LIN {X 0,Y 197.336,Z 414.265,A -85,B 0,C 180,E1 -21920.386,E2 -21920.386} C_VEL
LIN {X 0,Y 196.513,Z 412.639,A -85,B 0,C 180,E1 -21920.854,E2 -21920.854} C_VEL
LIN {X 0,Y 194.043,Z 410.71,A -85,B 0,C 180,E1 -21922.116,E2 -21922.116} C_VEL
LIN {X 0,Y 192.76,Z 408.182,A -85,B 0,C 180,E1 -21922.91,E2 -21922.91} C_VEL
LIN {X 0,Y 192.565,Z 407.12,A -85,B 0,C 180,E1 -21923.107,E2 -21923.107} C_VEL
LIN {X 0,Y 192.604,Z 407.109,A -85,B 0,C 180,E1 -21927.061,E2 -21927.061} C_VEL
LIN {X 0,Y 192.618,Z 407.106,A -85,B 0,C 180,E1 -21931.684,E2 -21931.684} C_VEL
LIN {X 0,Y 192.669,Z 407.096,A -85,B 0,C 180,E1 -21936.343,E2 -21936.343} C_VEL
LIN {X 0,Y 192.693,Z 407.092,A -85,B 0,C 180,E1 -21941.491,E2 -21941.491} C_VEL
LIN {X 0,Y 192.732,Z 407.089,A -85,B 0,C 180,E1 -21945.211,E2 -21945.211} C_VEL
LIN {X 0,Y 192.944,Z 407.006,A -85,B 0,C 180,E1 -21949.566,E2 -21949.566} C_VEL
LIN {X 0,Y 192.953,Z 407.069,A -85,B 0,C 180,E1 -21953.726,E2 -21953.726} C_VEL
LIN {X 0,Y 193.204,Z 407.021,A -85,B 0,C 180,E1 -21957.915,E2 -21957.915} C_VEL
LIN {X 0,Y 193.404,Z 407.012,A -85,B 0,C 180,E1 -21959.999,E2 -21959.999} C_VEL
LIN {X 0,Y 192.929,Z 407.057,A -85,B 0,C 180,E1 -21964.177,E2 -21964.177} C_VEL
LIN {X 0,Y 193.017,Z 407.052,A -85,B 0,C 180,E1 -21968.374,E2 -21968.374} C_VEL
LIN {X 0,Y 192.77,Z 407.094,A -85,B 0,C 180,E1 -21972.635,E2 -21972.635} C_VEL
LIN {X 0,Y 192.692,Z 407.097,A -85,B 0,C 180,E1 -21978.508,E2 -21978.508} C_VEL
LIN {X 0,Y 192.648,Z 407.204,A -85,B 0,C 180,E1 -21982.947,E2 -21982.947} C_VEL
LIN {X 0,Y 195.501,Z 414.864,A -85,B 0,C 180,E1 -21987.715,E2 -21987.715} C_VEL
LIN {X 0,Y 201.405,Z 424.233,A -85,B 0,C 180,E1 -21990.831,E2 -21990.831} C_VEL
LIN {X 0,Y 205.353,Z 430.73,A -85,B 0,C 180,E1 -21992.69,E2 -21992.69} C_VEL
LIN {X 0,Y 209.382,Z 437.854,A -85,B 0,C 180,E1 -21994.468,E2 -21994.468} C_VEL
LIN {X 0,Y 212.955,Z 444.606,A -85,B 0,C 180,E1 -21995.959,E2 -21995.959} C_VEL
LIN {X 0,Y 217.953,Z 454.685,A -85,B 0,C 180,E1 -21997.928,E2 -21997.928} C_VEL
LIN {X 0,Y 223.379,Z 466.674,A -85,B 0,C 180,E1 -21999.942,E2 -21999.942} C_VEL
LIN {X 0,Y 228.391,Z 479.658,A -85,B 0,C 180,E1 -22001.743,E2 -22001.743} C_VEL
LIN {X 0,Y 229.336,Z 493.154,A -85,B 0,C 180,E1 -22002.532,E2 -22002.532} C_VEL
LIN {X 0,Y 229.333,Z 498.97,A -85,B 0,C 180,E1 -22002.774,E2 -22002.774} C_VEL
LIN {X 0,Y 226.311,Z 518.591,A -85,B 0,C 180,E1 -22002.905,E2 -22002.905} C_VEL
LIN {X 0,Y 226.123,Z 524.463,A -85,B 0,C 180,E1 -22003.109,E2 -22003.109} C_VEL
LIN {X 0,Y 222.374,Z 588.724,A -85,B 0,C 180,E1 -22004.997,E2 -22004.997} C_VEL
LIN {X 0,Y 220.722,Z 604.246,A -85,B 0,C 180,E1 -22005.693,E2 -22005.693} C_VEL
LIN {X 0,Y 218.207,Z 619.257,A -85,B 0,C 180,E1 -22006.652,E2 -22006.652} C_VEL
LIN {X 0,Y 215.296,Z 632.891,A -85,B 0,C 180,E1 -22007.838,E2 -22007.838} C_VEL
LIN {X 0,Y 211.683,Z 646.439,A -85,B 0,C 180,E1 -22009.341,E2 -22009.341} C_VEL
LIN {X 0,Y 207.749,Z 658.936,A -85,B 0,C 180,E1 -22011.084,E2 -22011.084} C_VEL
LIN {X 0,Y 204.93,Z 667.258,A -85,B 0,C 180,E1 -22012.503,E2 -22012.503} C_VEL
LIN {X 0,Y 200.796,Z 679.406,A -85,B 0,C 180,E1 -22015.031,E2 -22015.031} C_VEL
LIN {X 0,Y 196.253,Z 691.345,A -85,B 0,C 180,E1 -22018.115,E2 -22018.115} C_VEL
LIN {X 0,Y 192.23,Z 702.077,A -85,B 0,C 180,E1 -22021.622,E2 -22021.622} C_VEL
LIN {X 0,Y 189.098,Z 711.051,A -85,B 0,C 180,E1 -22025.284,E2 -22025.284} C_VEL
LIN {X 0,Y 186.788,Z 718.548,A -85,B 0,C 180,E1 -22029.056,E2 -22029.056} C_VEL
LIN {X 0,Y 185.109,Z 725.529,A -85,B 0,C 180,E1 -22033.456,E2 -22033.456} C_VEL
LIN {X 0,Y 184.507,Z 731.031,A -85,B 0,C 180,E1 -22037.906,E2 -22037.906} C_VEL
LIN {X 0,Y 184.68,Z 734.604,A -85,B 0,C 180,E1 -22041.659,E2 -22041.659} C_VEL
LIN {X 0,Y 185.236,Z 737.321,A -85,B 0,C 180,E1 -22045.647,E2 -22045.647} C_VEL
LIN {X 0,Y 186.173,Z 739.099,A -85,B 0,C 180,E1 -22049.999,E2 -22049.999} C_VEL
LIN {X 0,Y 185.102,Z 739.29,A -85,B 0,C 180,E1 -22054.354,E2 -22054.354} C_VEL
LIN {X 0,Y 184.505,Z 738.486,A -85,B 0,C 180,E1 -22057.961,E2 -22057.961} C_VEL
LIN {X 0,Y 184.298,Z 735.96,A -85,B 0,C 180,E1 -22063.225,E2 -22063.225} C_VEL
LIN {X 0,Y 185.311,Z 732.569,A -85,B 0,C 180,E1 -22067.661,E2 -22067.661} C_VEL
LIN {X 0,Y 187.383,Z 727.977,A -85,B 0,C 180,E1 -22072.027,E2 -22072.027} C_VEL
LIN {X 0,Y 190.614,Z 722.095,A -85,B 0,C 180,E1 -22076.258,E2 -22076.258} C_VEL
LIN {X 0,Y 194.914,Z 714.773,A -85,B 0,C 180,E1 -22080.316,E2 -22080.316} C_VEL
LIN {X 0,Y 200.248,Z 705.81,A -85,B 0,C 180,E1 -22084.161,E2 -22084.161} C_VEL
LIN {X 0,Y 205.88,Z 696.435,A -85,B 0,C 180,E1 -22087.293,E2 -22087.293} C_VEL
LIN {X 0,Y 211.59,Z 686.323,A -85,B 0,C 180,E1 -22089.972,E2 -22089.972} C_VEL
LIN {X 0,Y 217.488,Z 674.798,A -85,B 0,C 180,E1 -22092.418,E2 -22092.418} C_VEL
LIN {X 0,Y 223.387,Z 662.521,A -85,B 0,C 180,E1 -22094.425,E2 -22094.425} C_VEL
LIN {X 0,Y 229.069,Z 649.104,A -85,B 0,C 180,E1 -22096.134,E2 -22096.134} C_VEL
LIN {X 0,Y 233.791,Z 636.023,A -85,B 0,C 180,E1 -22097.431,E2 -22097.431} C_VEL
LIN {X 0,Y 237.121,Z 625.222,A -85,B 0,C 180,E1 -22098.288,E2 -22098.288} C_VEL
LIN {X 0,Y 240.717,Z 610.446,A -85,B 0,C 180,E1 -22099.222,E2 -22099.222} C_VEL
LIN {X 0,Y 243.456,Z 595.214,A -85,B 0,C 180,E1 -22099.904,E2 -22099.904} C_VEL
LIN {X 0,Y 245.117,Z 579.442,A -85,B 0,C 180,E1 -22100.401,E2 -22100.401} C_VEL
LIN {X 0,Y 248.733,Z 529.136,A -85,B 0,C 180,E1 -22101.696,E2 -22101.696} C_VEL
LIN {X 0,Y 247.505,Z 504.831,A -85,B 0,C 180,E1 -22103.33,E2 -22103.33} C_VEL
LIN {X 0,Y 243.68,Z 494.924,A -85,B 0,C 180,E1 -22105.25,E2 -22105.25} C_VEL
LIN {X 0,Y 238.561,Z 483.088,A -85,B 0,C 180,E1 -22108.02,E2 -22108.02} C_VEL
LIN {X 0,Y 234.67,Z 475.032,A -85,B 0,C 180,E1 -22110.329,E2 -22110.329} C_VEL
LIN {X 0,Y 231.739,Z 469.172,A -85,B 0,C 180,E1 -22112.247,E2 -22112.247} C_VEL
LIN {X 0,Y 229.497,Z 464.737,A -85,B 0,C 180,E1 -22113.851,E2 -22113.851} C_VEL
LIN {X 0,Y 225.583,Z 457.444,A -85,B 0,C 180,E1 -22116.991,E2 -22116.991} C_VEL
LIN {X 0,Y 221.261,Z 449.476,A -85,B 0,C 180,E1 -22121.322,E2 -22121.322} C_VEL
LIN {X 0,Y 217.227,Z 441.913,A -85,B 0,C 180,E1 -22127.268,E2 -22127.268} C_VEL
LIN {X 0,Y 215.991,Z 439.112,A -85,B 0,C 180,E1 -22130.327,E2 -22130.327} C_VEL
LIN {X 0,Y 215.609,Z 438.486,A -85,B 0,C 180,E1 -22131.566,E2 -22131.566} C_VEL
LIN {X 0,Y 215.268,Z 438.207,A -85,B 0,C 180,E1 -22140,E2 -22140} C_VEL
LIN {X 0,Y 215.981,Z 438.646,A -85,B 0,C 180,E1 -22142.448,E2 -22142.448} C_VEL
LIN {X 0,Y 217.318,Z 441.615,A -85,B 0,C 180,E1 -22145.801,E2 -22145.801} C_VEL
LIN {X 0,Y 219.851,Z 444.129,A -85,B 0,C 180,E1 -22149.546,E2 -22149.546} C_VEL
LIN {X 0,Y 222.184,Z 447.842,A -85,B 0,C 180,E1 -22152.329,E2 -22152.329} C_VEL
LIN {X 0,Y 223.794,Z 449.538,A -85,B 0,C 180,E1 -22153.882,E2 -22153.882} C_VEL
LIN {X 0,Y 226.441,Z 453.257,A -85,B 0,C 180,E1 -22156.221,E2 -22156.221} C_VEL
LIN {X 0,Y 227.842,Z 455.259,A -85,B 0,C 180,E1 -22157.341,E2 -22157.341} C_VEL
LIN {X 0,Y 230.915,Z 459.466,A -85,B 0,C 180,E1 -22159.56,E2 -22159.56} C_VEL
LIN {X 0,Y 234.645,Z 464.805,A -85,B 0,C 180,E1 -22161.957,E2 -22161.957} C_VEL
LIN {X 0,Y 239.856,Z 472.69,A -85,B 0,C 180,E1 -22164.904,E2 -22164.904} C_VEL
LIN {X 0,Y 245.011,Z 481.125,A -85,B 0,C 180,E1 -22167.493,E2 -22167.493} C_VEL
LIN {X 0,Y 251.018,Z 491.976,A -85,B 0,C 180,E1 -22170.214,E2 -22170.214} C_VEL
LIN {X 0,Y 251.128,Z 492.964,A -85,B 0,C 180,E1 -22170.3,E2 -22170.3} C_VEL
LIN {X 0,Y 248.333,Z 535.874,A -85,B 0,C 180,E1 -22171.501,E2 -22171.501} C_VEL
LIN {X 0,Y 247.098,Z 551.646,A -85,B 0,C 180,E1 -22172.113,E2 -22172.113} C_VEL
LIN {X 0,Y 245.26,Z 565.698,A -85,B 0,C 180,E1 -22172.93,E2 -22172.93} C_VEL
LIN {X 0,Y 242.739,Z 578.445,A -85,B 0,C 180,E1 -22173.844,E2 -22173.844} C_VEL
LIN {X 0,Y 239.519,Z 591.832,A -85,B 0,C 180,E1 -22175.127,E2 -22175.127} C_VEL
LIN {X 0,Y 235.581,Z 604.678,A -85,B 0,C 180,E1 -22176.631,E2 -22176.631} C_VEL
LIN {X 0,Y 231.016,Z 617.087,A -85,B 0,C 180,E1 -22178.433,E2 -22178.433} C_VEL
LIN {X 0,Y 226.244,Z 628.273,A -85,B 0,C 180,E1 -22180.446,E2 -22180.446} C_VEL
LIN {X 0,Y 220.806,Z 639.452,A -85,B 0,C 180,E1 -22182.943,E2 -22182.943} C_VEL
LIN {X 0,Y 215.531,Z 649.063,A -85,B 0,C 180,E1 -22185.621,E2 -22185.621} C_VEL
LIN {X 0,Y 210.145,Z 657.847,A -85,B 0,C 180,E1 -22188.664,E2 -22188.664} C_VEL
LIN {X 0,Y 204.922,Z 665.612,A -85,B 0,C 180,E1 -22192.075,E2 -22192.075} C_VEL
LIN {X 0,Y 200.088,Z 672.19,A -85,B 0,C 180,E1 -22195.808,E2 -22195.808} C_VEL
LIN {X 0,Y 195.863,Z 677.52,A -85,B 0,C 180,E1 -22199.846,E2 -22199.846} C_VEL
LIN {X 0,Y 192.423,Z 681.468,A -85,B 0,C 180,E1 -22204.007,E2 -22204.007} C_VEL
LIN {X 0,Y 189.769,Z 684.161,A -85,B 0,C 180,E1 -22208.265,E2 -22208.265} C_VEL
LIN {X 0,Y 187.887,Z 685.683,A -85,B 0,C 180,E1 -22212.589,E2 -22212.589} C_VEL
LIN {X 0,Y 186.82,Z 686.072,A -85,B 0,C 180,E1 -22216.956,E2 -22216.956} C_VEL
LIN {X 0,Y 186.433,Z 685.316,A -85,B 0,C 180,E1 -22221.328,E2 -22221.328} C_VEL
LIN {X 0,Y 186.491,Z 683.481,A -85,B 0,C 180,E1 -22225.678,E2 -22225.678} C_VEL
LIN {X 0,Y 187.349,Z 680.499,A -85,B 0,C 180,E1 -22230.001,E2 -22230.001} C_VEL
LIN {X 0,Y 188.487,Z 677.504,A -85,B 0,C 180,E1 -22233.207,E2 -22233.207} C_VEL
LIN {X 0,Y 190.399,Z 672.384,A -85,B 0,C 180,E1 -22237.424,E2 -22237.424} C_VEL
LIN {X 0,Y 193.099,Z 665.862,A -85,B 0,C 180,E1 -22241.548,E2 -22241.548} C_VEL
LIN {X 0,Y 196.407,Z 657.773,A -85,B 0,C 180,E1 -22245.568,E2 -22245.568} C_VEL
LIN {X 0,Y 199.927,Z 649.129,A -85,B 0,C 180,E1 -22248.976,E2 -22248.976} C_VEL
LIN {X 0,Y 203.922,Z 638.764,A -85,B 0,C 180,E1 -22252.279,E2 -22252.279} C_VEL
LIN {X 0,Y 207.68,Z 628.116,A -85,B 0,C 180,E1 -22255.025,E2 -22255.025} C_VEL
LIN {X 0,Y 211.23,Z 616.543,A -85,B 0,C 180,E1 -22257.493,E2 -22257.493} C_VEL
LIN {X 0,Y 214.868,Z 603.829,A -85,B 0,C 180,E1 -22259.651,E2 -22259.651} C_VEL
LIN {X 0,Y 217.818,Z 591.526,A -85,B 0,C 180,E1 -22261.351,E2 -22261.351} C_VEL
LIN {X 0,Y 220.71,Z 577.159,A -85,B 0,C 180,E1 -22262.91,E2 -22262.91} C_VEL
LIN {X 0,Y 223.009,Z 562.117,A -85,B 0,C 180,E1 -22264.149,E2 -22264.149} C_VEL
LIN {X 0,Y 224.642,Z 546.333,A -85,B 0,C 180,E1 -22265.077,E2 -22265.077} C_VEL
LIN {X 0,Y 225.602,Z 526.89,A -85,B 0,C 180,E1 -22265.822,E2 -22265.822} C_VEL
LIN {X 0,Y 228.471,Z 474.221,A -85,B 0,C 180,E1 -22267.384,E2 -22267.384} C_VEL
LIN {X 0,Y 221.357,Z 460.213,A -85,B 0,C 180,E1 -22269.795,E2 -22269.795} C_VEL
LIN {X 0,Y 214.974,Z 449.162,A -85,B 0,C 180,E1 -22272.118,E2 -22272.118} C_VEL
LIN {X 0,Y 209.036,Z 439.887,A -85,B 0,C 180,E1 -22274.458,E2 -22274.458} C_VEL
LIN {X 0,Y 203.255,Z 431.624,A -85,B 0,C 180,E1 -22276.947,E2 -22276.947} C_VEL
LIN {X 0,Y 200.324,Z 427.619,A -85,B 0,C 180,E1 -22278.311,E2 -22278.311} C_VEL
LIN {X 0,Y 197.158,Z 423.413,A -85,B 0,C 180,E1 -22279.877,E2 -22279.877} C_VEL
LIN {X 0,Y 194.456,Z 419.981,A -85,B 0,C 180,E1 -22281.295,E2 -22281.295} C_VEL
LIN {X 0,Y 193.679,Z 418.8,A -85,B 0,C 180,E1 -22281.734,E2 -22281.734} C_VEL
LIN {X 0,Y 191.072,Z 416.164,A -85,B 0,C 180,E1 -22283.178,E2 -22283.178} C_VEL
LIN {X 0,Y 189.815,Z 413.672,A -85,B 0,C 180,E1 -22284,E2 -22284} C_VEL
LIN {X 0,Y 187.19,Z 411.797,A -85,B 0,C 180,E1 -22285.561,E2 -22285.561} C_VEL
LIN {X 0,Y 185.935,Z 409.573,A -85,B 0,C 180,E1 -22286.46,E2 -22286.46} C_VEL
LIN {X 0,Y 185.564,Z 407.985,A -85,B 0,C 180,E1 -22286.894,E2 -22286.894} C_VEL
LIN {X 0,Y 185.546,Z 407.986,A -85,B 0,C 180,E1 -22290.595,E2 -22290.595} C_VEL
LIN {X 0,Y 185.58,Z 407.98,A -85,B 0,C 180,E1 -22295.381,E2 -22295.381} C_VEL
LIN {X 0,Y 185.624,Z 407.972,A -85,B 0,C 180,E1 -22301.178,E2 -22301.178} C_VEL
LIN {X 0,Y 185.661,Z 407.978,A -85,B 0,C 180,E1 -22304.634,E2 -22304.634} C_VEL
LIN {X 0,Y 185.886,Z 407.883,A -85,B 0,C 180,E1 -22309.419,E2 -22309.419} C_VEL
LIN {X 0,Y 185.919,Z 407.939,A -85,B 0,C 180,E1 -22313.488,E2 -22313.488} C_VEL
LIN {X 0,Y 186.37,Z 407.888,A -85,B 0,C 180,E1 -22319.999,E2 -22319.999} C_VEL
LIN {X 0,Y 185.877,Z 407.936,A -85,B 0,C 180,E1 -22324.336,E2 -22324.336} C_VEL
LIN {X 0,Y 185.968,Z 407.928,A -85,B 0,C 180,E1 -22328.694,E2 -22328.694} C_VEL
LIN {X 0,Y 185.694,Z 407.969,A -85,B 0,C 180,E1 -22333.125,E2 -22333.125} C_VEL
LIN {X 0,Y 185.622,Z 407.977,A -85,B 0,C 180,E1 -22338.82,E2 -22338.82} C_VEL
LIN {X 0,Y 185.538,Z 408.144,A -85,B 0,C 180,E1 -22340.221,E2 -22340.221} C_VEL
LIN {X 0,Y 187.482,Z 412.98,A -85,B 0,C 180,E1 -22343.617,E2 -22343.617} C_VEL
LIN {X 0,Y 191.023,Z 418.479,A -85,B 0,C 180,E1 -22345.885,E2 -22345.885} C_VEL
LIN {X 0,Y 193.755,Z 422.546,A -85,B 0,C 180,E1 -22347.473,E2 -22347.473} C_VEL
LIN {X 0,Y 198.157,Z 429.503,A -85,B 0,C 180,E1 -22349.844,E2 -22349.844} C_VEL
LIN {X 0,Y 202.324,Z 436.64,A -85,B 0,C 180,E1 -22351.913,E2 -22351.913} C_VEL
LIN {X 0,Y 206.428,Z 444.154,A -85,B 0,C 180,E1 -22353.809,E2 -22353.809} C_VEL
LIN {X 0,Y 211.239,Z 453.61,A -85,B 0,C 180,E1 -22355.882,E2 -22355.882} C_VEL
LIN {X 0,Y 217.487,Z 467.235,A -85,B 0,C 180,E1 -22358.392,E2 -22358.392} C_VEL
LIN {X 0,Y 223.323,Z 481.972,A -85,B 0,C 180,E1 -22360.609,E2 -22360.609} C_VEL
LIN {X 0,Y 226.123,Z 524.463,A -85,B 0,C 180,E1 -22363.109,E2 -22363.109} C_VEL
LIN {X 0,Y 225.98,Z 528.334,A -85,B 0,C 180,E1 -22363.239,E2 -22363.239} C_VEL
LIN {X 0,Y 225.302,Z 532.197,A -85,B 0,C 180,E1 -22363.247,E2 -22363.247} C_VEL
LIN {X 0,Y 223.029,Z 539.775,A -85,B 0,C 180,E1 -22363.046,E2 -22363.046} C_VEL
LIN {X 0,Y 220.022,Z 549.308,A -85,B 0,C 180,E1 -22362.751,E2 -22362.751} C_VEL
LIN {X 0,Y 219.083,Z 555.205,A -85,B 0,C 180,E1 -22362.785,E2 -22362.785} C_VEL
LIN {X 0,Y 216.861,Z 590.046,A -85,B 0,C 180,E1 -22363.838,E2 -22363.838} C_VEL
LIN {X 0,Y 214.982,Z 605.773,A -85,B 0,C 180,E1 -22364.598,E2 -22364.598} C_VEL
LIN {X 0,Y 212.04,Z 621.914,A -85,B 0,C 180,E1 -22365.725,E2 -22365.725} C_VEL
LIN {X 0,Y 208.816,Z 635.791,A -85,B 0,C 180,E1 -22367.036,E2 -22367.036} C_VEL
LIN {X 0,Y 204.781,Z 649.335,A -85,B 0,C 180,E1 -22368.651,E2 -22368.651} C_VEL
LIN {X 0,Y 200.874,Z 660.933,A -85,B 0,C 180,E1 -22370.416,E2 -22370.416} C_VEL
LIN {X 0,Y 196.388,Z 673.605,A -85,B 0,C 180,E1 -22372.851,E2 -22372.851} C_VEL
LIN {X 0,Y 192.264,Z 684.575,A -85,B 0,C 180,E1 -22375.488,E2 -22375.488} C_VEL
LIN {X 0,Y 188.25,Z 694.74,A -85,B 0,C 180,E1 -22378.489,E2 -22378.489} C_VEL
LIN {X 0,Y 184.371,Z 704.741,A -85,B 0,C 180,E1 -22382.163,E2 -22382.163} C_VEL
LIN {X 0,Y 181.365,Z 713.116,A -85,B 0,C 180,E1 -22385.991,E2 -22385.991} C_VEL
LIN {X 0,Y 179.025,Z 720.844,A -85,B 0,C 180,E1 -22390.418,E2 -22390.418} C_VEL
LIN {X 0,Y 177.69,Z 727.245,A -85,B 0,C 180,E1 -22395.102,E2 -22395.102} C_VEL
LIN {X 0,Y 177.483,Z 732.108,A -85,B 0,C 180,E1 -22399.735,E2 -22399.735} C_VEL
LIN {X 0,Y 177.816,Z 734.823,A -85,B 0,C 180,E1 -22403.19,E2 -22403.19} C_VEL
LIN {X 0,Y 178.165,Z 736.223,A -85,B 0,C 180,E1 -22405.474,E2 -22405.474} C_VEL
LIN {X 0,Y 179.128,Z 738.05,A -85,B 0,C 180,E1 -22409.999,E2 -22409.999} C_VEL
LIN {X 0,Y 178.03,Z 738.272,A -85,B 0,C 180,E1 -22414.527,E2 -22414.527} C_VEL
LIN {X 0,Y 177.284,Z 737.215,A -85,B 0,C 180,E1 -22419.123,E2 -22419.123} C_VEL
LIN {X 0,Y 177.307,Z 734.997,A -85,B 0,C 180,E1 -22423.757,E2 -22423.757} C_VEL
LIN {X 0,Y 178.463,Z 731.648,A -85,B 0,C 180,E1 -22428.362,E2 -22428.362} C_VEL
LIN {X 0,Y 180.707,Z 727.101,A -85,B 0,C 180,E1 -22432.886,E2 -22432.886} C_VEL
LIN {X 0,Y 184.171,Z 721.27,A -85,B 0,C 180,E1 -22437.251,E2 -22437.251} C_VEL
LIN {X 0,Y 188.738,Z 714.001,A -85,B 0,C 180,E1 -22441.419,E2 -22441.419} C_VEL
LIN {X 0,Y 194.323,Z 705.106,A -85,B 0,C 180,E1 -22445.355,E2 -22445.355} C_VEL
LIN {X 0,Y 200.228,Z 695.794,A -85,B 0,C 180,E1 -22448.535,E2 -22448.535} C_VEL
LIN {X 0,Y 206.518,Z 685.09,A -85,B 0,C 180,E1 -22451.414,E2 -22451.414} C_VEL
LIN {X 0,Y 212.81,Z 673.316,A -85,B 0,C 180,E1 -22453.907,E2 -22453.907} C_VEL
LIN {X 0,Y 218.917,Z 660.956,A -85,B 0,C 180,E1 -22455.913,E2 -22455.913} C_VEL
LIN {X 0,Y 224.808,Z 647.432,A -85,B 0,C 180,E1 -22457.607,E2 -22457.607} C_VEL
LIN {X 0,Y 229.675,Z 634.206,A -85,B 0,C 180,E1 -22458.893,E2 -22458.893} C_VEL
LIN {X 0,Y 232.766,Z 624.323,A -85,B 0,C 180,E1 -22459.672,E2 -22459.672} C_VEL
LIN {X 0,Y 236.474,Z 609.599,A -85,B 0,C 180,E1 -22460.596,E2 -22460.596} C_VEL
LIN {X 0,Y 239.295,Z 594.464,A -85,B 0,C 180,E1 -22461.27,E2 -22461.27} C_VEL
LIN {X 0,Y 240.989,Z 578.874,A -85,B 0,C 180,E1 -22461.772,E2 -22461.772} C_VEL
LIN {X 0,Y 244.611,Z 529.708,A -85,B 0,C 180,E1 -22463.052,E2 -22463.052} C_VEL
LIN {X 0,Y 243.587,Z 507.937,A -85,B 0,C 180,E1 -22464.574,E2 -22464.574} C_VEL
LIN {X 0,Y 239.63,Z 497.574,A -85,B 0,C 180,E1 -22466.701,E2 -22466.701} C_VEL
LIN {X 0,Y 235.094,Z 487.034,A -85,B 0,C 180,E1 -22469.332,E2 -22469.332} C_VEL
LIN {X 0,Y 231.593,Z 479.41,A -85,B 0,C 180,E1 -22471.583,E2 -22471.583} C_VEL
LIN {X 0,Y 227.566,Z 471.05,A -85,B 0,C 180,E1 -22474.505,E2 -22474.505} C_VEL
LIN {X 0,Y 223.624,Z 463.448,A -85,B 0,C 180,E1 -22477.844,E2 -22477.844} C_VEL
LIN {X 0,Y 219.825,Z 456.076,A -85,B 0,C 180,E1 -22481.894,E2 -22481.894} C_VEL
LIN {X 0,Y 216.002,Z 448.548,A -85,B 0,C 180,E1 -22487.925,E2 -22487.925} C_VEL
LIN {X 0,Y 214.956,Z 445.866,A -85,B 0,C 180,E1 -22490.829,E2 -22490.829} C_VEL
LIN {X 0,Y 214.485,Z 445.429,A -85,B 0,C 180,E1 -22492.469,E2 -22492.469} C_VEL
LIN {X 0,Y 214.397,Z 445.241,A -85,B 0,C 180,E1 -22500,E2 -22500} C_VEL
LIN {X 0,Y 215.002,Z 445.658,A -85,B 0,C 180,E1 -22502.167,E2 -22502.167} C_VEL
LIN {X 0,Y 216.558,Z 448.989,A -85,B 0,C 180,E1 -22506.055,E2 -22506.055} C_VEL
LIN {X 0,Y 218.648,Z 451.068,A -85,B 0,C 180,E1 -22509.176,E2 -22509.176} C_VEL
LIN {X 0,Y 220.998,Z 454.781,A -85,B 0,C 180,E1 -22512.061,E2 -22512.061} C_VEL
LIN {X 0,Y 222.377,Z 456.359,A -85,B 0,C 180,E1 -22513.443,E2 -22513.443} C_VEL
LIN {X 0,Y 225.036,Z 460.073,A -85,B 0,C 180,E1 -22515.859,E2 -22515.859} C_VEL
LIN {X 0,Y 229.114,Z 466.026,A -85,B 0,C 180,E1 -22519.022,E2 -22519.022} C_VEL
LIN {X 0,Y 232.956,Z 471.671,A -85,B 0,C 180,E1 -22521.573,E2 -22521.573} C_VEL
LIN {X 0,Y 238.126,Z 479.766,A -85,B 0,C 180,E1 -22524.58,E2 -22524.58} C_VEL
LIN {X 0,Y 243.753,Z 489.467,A -85,B 0,C 180,E1 -22527.473,E2 -22527.473} C_VEL
LIN {X 0,Y 246.976,Z 495.537,A -85,B 0,C 180,E1 -22528.995,E2 -22528.995} C_VEL
LIN {X 0,Y 243.863,Z 542.221,A -85,B 0,C 180,E1 -22530.357,E2 -22530.357} C_VEL
LIN {X 0,Y 242.371,Z 557.22,A -85,B 0,C 180,E1 -22531.027,E2 -22531.027} C_VEL
LIN {X 0,Y 240.104,Z 571.442,A -85,B 0,C 180,E1 -22531.917,E2 -22531.917} C_VEL
LIN {X 0,Y 237.431,Z 583.821,A -85,B 0,C 180,E1 -22532.912,E2 -22532.912} C_VEL
LIN {X 0,Y 233.86,Z 596.961,A -85,B 0,C 180,E1 -22534.269,E2 -22534.269} C_VEL
LIN {X 0,Y 229.54,Z 609.658,A -85,B 0,C 180,E1 -22535.868,E2 -22535.868} C_VEL
LIN {X 0,Y 224.561,Z 621.983,A -85,B 0,C 180,E1 -22537.795,E2 -22537.795} C_VEL
LIN {X 0,Y 219.188,Z 633.557,A -85,B 0,C 180,E1 -22540.071,E2 -22540.071} C_VEL
LIN {X 0,Y 214.137,Z 643.16,A -85,B 0,C 180,E1 -22542.403,E2 -22542.403} C_VEL
LIN {X 0,Y 208,Z 653.459,A -85,B 0,C 180,E1 -22545.504,E2 -22545.504} C_VEL
LIN {X 0,Y 202.461,Z 661.855,A -85,B 0,C 180,E1 -22548.737,E2 -22548.737} C_VEL
LIN {X 0,Y 196.746,Z 669.67,A -85,B 0,C 180,E1 -22552.611,E2 -22552.611} C_VEL
LIN {X 0,Y 191.835,Z 675.82,A -85,B 0,C 180,E1 -22556.667,E2 -22556.667} C_VEL
LIN {X 0,Y 187.732,Z 680.505,A -85,B 0,C 180,E1 -22560.88,E2 -22560.88} C_VEL
LIN {X 0,Y 184.436,Z 683.873,A -85,B 0,C 180,E1 -22565.22,E2 -22565.22} C_VEL
LIN {X 0,Y 181.954,Z 686.031,A -85,B 0,C 180,E1 -22569.659,E2 -22569.659} C_VEL
LIN {X 0,Y 180.364,Z 687.034,A -85,B 0,C 180,E1 -22574.173,E2 -22574.173} C_VEL
LIN {X 0,Y 179.568,Z 686.877,A -85,B 0,C 180,E1 -22578.716,E2 -22578.716} C_VEL
LIN {X 0,Y 179.278,Z 685.637,A -85,B 0,C 180,E1 -22583.247,E2 -22583.247} C_VEL
LIN {X 0,Y 179.811,Z 683.274,A -85,B 0,C 180,E1 -22587.761,E2 -22587.761} C_VEL
LIN {X 0,Y 181.094,Z 679.751,A -85,B 0,C 180,E1 -22592.225,E2 -22592.225} C_VEL
LIN {X 0,Y 182.852,Z 675.04,A -85,B 0,C 180,E1 -22596.622,E2 -22596.622} C_VEL
LIN {X 0,Y 185.471,Z 668.954,A -85,B 0,C 180,E1 -22600.922,E2 -22600.922} C_VEL
LIN {X 0,Y 188.75,Z 661.344,A -85,B 0,C 180,E1 -22605.109,E2 -22605.109} C_VEL
LIN {X 0,Y 192.239,Z 653.244,A -85,B 0,C 180,E1 -22608.657,E2 -22608.657} C_VEL
LIN {X 0,Y 196.287,Z 643.492,A -85,B 0,C 180,E1 -22612.083,E2 -22612.083} C_VEL
LIN {X 0,Y 200.077,Z 633.551,A -85,B 0,C 180,E1 -22614.931,E2 -22614.931} C_VEL
LIN {X 0,Y 204.065,Z 621.734,A -85,B 0,C 180,E1 -22617.706,E2 -22617.706} C_VEL
LIN {X 0,Y 207.746,Z 609.857,A -85,B 0,C 180,E1 -22619.933,E2 -22619.933} C_VEL
LIN {X 0,Y 211.17,Z 596.985,A -85,B 0,C 180,E1 -22621.893,E2 -22621.893} C_VEL
LIN {X 0,Y 213.896,Z 584.753,A -85,B 0,C 180,E1 -22623.391,E2 -22623.391} C_VEL
LIN {X 0,Y 216.527,Z 570.473,A -85,B 0,C 180,E1 -22624.753,E2 -22624.753} C_VEL
LIN {X 0,Y 218.604,Z 555.001,A -85,B 0,C 180,E1 -22625.846,E2 -22625.846} C_VEL
LIN {X 0,Y 219.823,Z 539.23,A -85,B 0,C 180,E1 -22626.622,E2 -22626.622} C_VEL
LIN {X 0,Y 221.989,Z 497.517,A -85,B 0,C 180,E1 -22627.952,E2 -22627.952} C_VEL
LIN {X 0,Y 223.127,Z 476.551,A -85,B 0,C 180,E1 -22628.596,E2 -22628.596} C_VEL
LIN {X 0,Y 216.41,Z 463.273,A -85,B 0,C 180,E1 -22631.016,E2 -22631.016} C_VEL
LIN {X 0,Y 210.286,Z 452.588,A -85,B 0,C 180,E1 -22633.386,E2 -22633.386} C_VEL
LIN {X 0,Y 203.431,Z 441.916,A -85,B 0,C 180,E1 -22636.294,E2 -22636.294} C_VEL
LIN {X 0,Y 197.488,Z 433.534,A -85,B 0,C 180,E1 -22639.099,E2 -22639.099} C_VEL
LIN {X 0,Y 194.181,Z 429.156,A -85,B 0,C 180,E1 -22640.808,E2 -22640.808} C_VEL
LIN {X 0,Y 190.972,Z 424.876,A -85,B 0,C 180,E1 -22642.605,E2 -22642.605} C_VEL
LIN {X 0,Y 188.282,Z 421.747,A -85,B 0,C 180,E1 -22644.2,E2 -22644.2} C_VEL
LIN {X 0,Y 187.156,Z 419.947,A -85,B 0,C 180,E1 -22644.943,E2 -22644.943} C_VEL
LIN {X 0,Y 184.572,Z 417.543,A -85,B 0,C 180,E1 -22646.609,E2 -22646.609} C_VEL
LIN {X 0,Y 183.022,Z 414.636,A -85,B 0,C 180,E1 -22647.805,E2 -22647.805} C_VEL
LIN {X 0,Y 180.397,Z 412.926,A -85,B 0,C 180,E1 -22649.699,E2 -22649.699} C_VEL
LIN {X 0,Y 178.783,Z 410.261,A -85,B 0,C 180,E1 -22651.126,E2 -22651.126} C_VEL
LIN {X 0,Y 178.468,Z 408.868,A -85,B 0,C 180,E1 -22651.605,E2 -22651.605} C_VEL
LIN {X 0,Y 178.515,Z 408.863,A -85,B 0,C 180,E1 -22654.889,E2 -22654.889} C_VEL
LIN {X 0,Y 178.606,Z 408.847,A -85,B 0,C 180,E1 -22661.651,E2 -22661.651} C_VEL
LIN {X 0,Y 178.638,Z 408.813,A -85,B 0,C 180,E1 -22666.346,E2 -22666.346} C_VEL
LIN {X 0,Y 178.898,Z 408.762,A -85,B 0,C 180,E1 -22670.958,E2 -22670.958} C_VEL
LIN {X 0,Y 178.811,Z 408.832,A -85,B 0,C 180,E1 -22675.491,E2 -22675.491} C_VEL
LIN {X 0,Y 179.335,Z 408.764,A -85,B 0,C 180,E1 -22679.999,E2 -22679.999} C_VEL
LIN {X 0,Y 178.826,Z 408.814,A -85,B 0,C 180,E1 -22684.508,E2 -22684.508} C_VEL
LIN {X 0,Y 178.899,Z 408.807,A -85,B 0,C 180,E1 -22689.04,E2 -22689.04} C_VEL
LIN {X 0,Y 178.621,Z 408.847,A -85,B 0,C 180,E1 -22693.654,E2 -22693.654} C_VEL
LIN {X 0,Y 178.6,Z 408.92,A -85,B 0,C 180,E1 -22697.017,E2 -22697.017} C_VEL
LIN {X 0,Y 178.899,Z 410.193,A -85,B 0,C 180,E1 -22697.873,E2 -22697.873} C_VEL
LIN {X 0,Y 180.298,Z 412.718,A -85,B 0,C 180,E1 -22699.129,E2 -22699.129} C_VEL
LIN {X 0,Y 181.597,Z 414.391,A -85,B 0,C 180,E1 -22700.171,E2 -22700.171} C_VEL
LIN {X 0,Y 185.189,Z 419.283,A -85,B 0,C 180,E1 -22702.817,E2 -22702.817} C_VEL
LIN {X 0,Y 188.765,Z 424.833,A -85,B 0,C 180,E1 -22705.203,E2 -22705.203} C_VEL
LIN {X 0,Y 194.451,Z 433.875,A -85,B 0,C 180,E1 -22708.539,E2 -22708.539} C_VEL
LIN {X 0,Y 199.007,Z 441.919,A -85,B 0,C 180,E1 -22710.947,E2 -22710.947} C_VEL
LIN {X 0,Y 204.146,Z 451.573,A -85,B 0,C 180,E1 -22713.423,E2 -22713.423} C_VEL
LIN {X 0,Y 209.79,Z 463.628,A -85,B 0,C 180,E1 -22715.941,E2 -22715.941} C_VEL
LIN {X 0,Y 214.854,Z 475.479,A -85,B 0,C 180,E1 -22718.043,E2 -22718.043} C_VEL
LIN {X 0,Y 218.362,Z 484.747,A -85,B 0,C 180,E1 -22719.449,E2 -22719.449} C_VEL
LIN {X 0,Y 220.878,Z 526.625,A -85,B 0,C 180,E1 -22721.969,E2 -22721.969} C_VEL
LIN {X 0,Y 219.083,Z 555.205,A -85,B 0,C 180,E1 -22722.785,E2 -22722.785} C_VEL
LIN {X 0,Y 218.258,Z 561.052,A -85,B 0,C 180,E1 -22722.84,E2 -22722.84} C_VEL
LIN {X 0,Y 212.867,Z 580.072,A -85,B 0,C 180,E1 -22722.377,E2 -22722.377} C_VEL
LIN {X 0,Y 211.906,Z 585.907,A -85,B 0,C 180,E1 -22722.442,E2 -22722.442} C_VEL
LIN {X 0,Y 210.126,Z 601.77,A -85,B 0,C 180,E1 -22723.152,E2 -22723.152} C_VEL
LIN {X 0,Y 207.507,Z 616.942,A -85,B 0,C 180,E1 -22724.144,E2 -22724.144} C_VEL
LIN {X 0,Y 204.089,Z 631.635,A -85,B 0,C 180,E1 -22725.442,E2 -22725.442} C_VEL
LIN {X 0,Y 200.025,Z 645.842,A -85,B 0,C 180,E1 -22727.098,E2 -22727.098} C_VEL
LIN {X 0,Y 195.79,Z 658.217,A -85,B 0,C 180,E1 -22728.921,E2 -22728.921} C_VEL
LIN {X 0,Y 192.807,Z 666.288,A -85,B 0,C 180,E1 -22730.365,E2 -22730.365} C_VEL
LIN {X 0,Y 188.34,Z 678.257,A -85,B 0,C 180,E1 -22733.007,E2 -22733.007} C_VEL
LIN {X 0,Y 183.459,Z 690.054,A -85,B 0,C 180,E1 -22736.257,E2 -22736.257} C_VEL
LIN {X 0,Y 179.668,Z 699.255,A -85,B 0,C 180,E1 -22739.435,E2 -22739.435} C_VEL
LIN {X 0,Y 176.04,Z 708.348,A -85,B 0,C 180,E1 -22743.312,E2 -22743.312} C_VEL
LIN {X 0,Y 173.349,Z 715.965,A -85,B 0,C 180,E1 -22747.346,E2 -22747.346} C_VEL
LIN {X 0,Y 171.315,Z 723.057,A -85,B 0,C 180,E1 -22752.08,E2 -22752.08} C_VEL
LIN {X 0,Y 170.418,Z 728.658,A -85,B 0,C 180,E1 -22756.89,E2 -22756.89} C_VEL
LIN {X 0,Y 170.558,Z 732.705,A -85,B 0,C 180,E1 -22761.468,E2 -22761.468} C_VEL
LIN {X 0,Y 171.09,Z 735.123,A -85,B 0,C 180,E1 -22765.287,E2 -22765.287} C_VEL
LIN {X 0,Y 172.081,Z 737,A -85,B 0,C 180,E1 -22769.999,E2 -22769.999} C_VEL
LIN {X 0,Y 170.955,Z 737.245,A -85,B 0,C 180,E1 -22774.715,E2 -22774.715} C_VEL
LIN {X 0,Y 170.215,Z 736.212,A -85,B 0,C 180,E1 -22779.505,E2 -22779.505} C_VEL
LIN {X 0,Y 170.307,Z 734.029,A -85,B 0,C 180,E1 -22784.334,E2 -22784.334} C_VEL
LIN {X 0,Y 171.984,Z 730,A -85,B 0,C 180,E1 -22789.97,E2 -22789.97} C_VEL
LIN {X 0,Y 174.885,Z 724.872,A -85,B 0,C 180,E1 -22794.957,E2 -22794.957} C_VEL
LIN {X 0,Y 178.854,Z 718.728,A -85,B 0,C 180,E1 -22799.417,E2 -22799.417} C_VEL
LIN {X 0,Y 184.002,Z 711.134,A -85,B 0,C 180,E1 -22803.628,E2 -22803.628} C_VEL
LIN {X 0,Y 189.322,Z 703.136,A -85,B 0,C 180,E1 -22807.099,E2 -22807.099} C_VEL
LIN {X 0,Y 195.558,Z 693.66,A -85,B 0,C 180,E1 -22810.305,E2 -22810.305} C_VEL
LIN {X 0,Y 201.41,Z 684.08,A -85,B 0,C 180,E1 -22812.881,E2 -22812.881} C_VEL
LIN {X 0,Y 208.296,Z 671.822,A -85,B 0,C 180,E1 -22815.458,E2 -22815.458} C_VEL
LIN {X 0,Y 214.618,Z 659.387,A -85,B 0,C 180,E1 -22817.457,E2 -22817.457} C_VEL
LIN {X 0,Y 220.702,Z 645.747,A -85,B 0,C 180,E1 -22819.135,E2 -22819.135} C_VEL
LIN {X 0,Y 225.676,Z 632.393,A -85,B 0,C 180,E1 -22820.42,E2 -22820.42} C_VEL
LIN {X 0,Y 230.163,Z 617.796,A -85,B 0,C 180,E1 -22821.483,E2 -22821.483} C_VEL
LIN {X 0,Y 233.673,Z 602.692,A -85,B 0,C 180,E1 -22822.312,E2 -22822.312} C_VEL
LIN {X 0,Y 236.13,Z 586.994,A -85,B 0,C 180,E1 -22822.939,E2 -22822.939} C_VEL
LIN {X 0,Y 240.29,Z 536.089,A -85,B 0,C 180,E1 -22824.269,E2 -22824.269} C_VEL
LIN {X 0,Y 240.637,Z 530.537,A -85,B 0,C 180,E1 -22824.443,E2 -22824.443} C_VEL
LIN {X 0,Y 239.871,Z 511.364,A -85,B 0,C 180,E1 -22825.807,E2 -22825.807} C_VEL
LIN {X 0,Y 236.12,Z 501.384,A -85,B 0,C 180,E1 -22827.96,E2 -22827.96} C_VEL
LIN {X 0,Y 232.288,Z 492.11,A -85,B 0,C 180,E1 -22830.343,E2 -22830.343} C_VEL
LIN {X 0,Y 229.134,Z 484.964,A -85,B 0,C 180,E1 -22832.502,E2 -22832.502} C_VEL
LIN {X 0,Y 225.332,Z 476.766,A -85,B 0,C 180,E1 -22835.437,E2 -22835.437} C_VEL
LIN {X 0,Y 221.788,Z 469.584,A -85,B 0,C 180,E1 -22838.644,E2 -22838.644} C_VEL
LIN {X 0,Y 218.304,Z 462.475,A -85,B 0,C 180,E1 -22842.613,E2 -22842.613} C_VEL
LIN {X 0,Y 214.994,Z 455.501,A -85,B 0,C 180,E1 -22848.174,E2 -22848.174} C_VEL
LIN {X 0,Y 213.976,Z 452.858,A -85,B 0,C 180,E1 -22851.144,E2 -22851.144} C_VEL
LIN {X 0,Y 213.62,Z 452.48,A -85,B 0,C 180,E1 -22852.439,E2 -22852.439} C_VEL
LIN {X 0,Y 213.525,Z 452.29,A -85,B 0,C 180,E1 -22860,E2 -22860} C_VEL
LIN {X 0,Y 214.065,Z 452.797,A -85,B 0,C 180,E1 -22862.029,E2 -22862.029} C_VEL
LIN {X 0,Y 215.764,Z 456.241,A -85,B 0,C 180,E1 -22866.23,E2 -22866.23} C_VEL
LIN {X 0,Y 217.445,Z 457.981,A -85,B 0,C 180,E1 -22868.788,E2 -22868.788} C_VEL
LIN {X 0,Y 219.83,Z 461.744,A -85,B 0,C 180,E1 -22871.804,E2 -22871.804} C_VEL
LIN {X 0,Y 220.964,Z 463.108,A -85,B 0,C 180,E1 -22872.982,E2 -22872.982} C_VEL
LIN {X 0,Y 223.431,Z 466.672,A -85,B 0,C 180,E1 -22875.318,E2 -22875.318} C_VEL
LIN {X 0,Y 227.408,Z 472.677,A -85,B 0,C 180,E1 -22878.527,E2 -22878.527} C_VEL
LIN {X 0,Y 231.445,Z 478.791,A -85,B 0,C 180,E1 -22881.29,E2 -22881.29} C_VEL
LIN {X 0,Y 236.422,Z 487.026,A -85,B 0,C 180,E1 -22884.272,E2 -22884.272} C_VEL
LIN {X 0,Y 241.203,Z 495.598,A -85,B 0,C 180,E1 -22886.819,E2 -22886.819} C_VEL
LIN {X 0,Y 242.847,Z 498.793,A -85,B 0,C 180,E1 -22887.642,E2 -22887.642} C_VEL
LIN {X 0,Y 239.578,Z 547.046,A -85,B 0,C 180,E1 -22889.127,E2 -22889.127} C_VEL
LIN {X 0,Y 237.791,Z 562.05,A -85,B 0,C 180,E1 -22889.873,E2 -22889.873} C_VEL
LIN {X 0,Y 235.456,Z 574.667,A -85,B 0,C 180,E1 -22890.699,E2 -22890.699} C_VEL
LIN {X 0,Y 231.957,Z 589.303,A -85,B 0,C 180,E1 -22891.97,E2 -22891.97} C_VEL
LIN {X 0,Y 227.695,Z 603.359,A -85,B 0,C 180,E1 -22893.556,E2 -22893.556} C_VEL
LIN {X 0,Y 222.841,Z 616.088,A -85,B 0,C 180,E1 -22895.312,E2 -22895.312} C_VEL
LIN {X 0,Y 217.647,Z 627.764,A -85,B 0,C 180,E1 -22897.334,E2 -22897.334} C_VEL
LIN {X 0,Y 212.069,Z 638.727,A -85,B 0,C 180,E1 -22899.702,E2 -22899.702} C_VEL
LIN {X 0,Y 206.453,Z 648.47,A -85,B 0,C 180,E1 -22902.309,E2 -22902.309} C_VEL
LIN {X 0,Y 200.395,Z 657.839,A -85,B 0,C 180,E1 -22905.462,E2 -22905.462} C_VEL
LIN {X 0,Y 195.518,Z 664.68,A -85,B 0,C 180,E1 -22908.321,E2 -22908.321} C_VEL
LIN {X 0,Y 189.683,Z 672.131,A -85,B 0,C 180,E1 -22912.315,E2 -22912.315} C_VEL
LIN {X 0,Y 184.591,Z 678.085,A -85,B 0,C 180,E1 -22916.624,E2 -22916.624} C_VEL
LIN {X 0,Y 181.474,Z 681.354,A -85,B 0,C 180,E1 -22919.773,E2 -22919.773} C_VEL
LIN {X 0,Y 177.944,Z 684.779,A -85,B 0,C 180,E1 -22924.251,E2 -22924.251} C_VEL
LIN {X 0,Y 175.256,Z 686.993,A -85,B 0,C 180,E1 -22928.845,E2 -22928.845} C_VEL
LIN {X 0,Y 173.5,Z 688.04,A -85,B 0,C 180,E1 -22933.529,E2 -22933.529} C_VEL
LIN {X 0,Y 172.594,Z 687.916,A -85,B 0,C 180,E1 -22938.254,E2 -22938.254} C_VEL
LIN {X 0,Y 172.251,Z 686.726,A -85,B 0,C 180,E1 -22942.97,E2 -22942.97} C_VEL
LIN {X 0,Y 172.753,Z 684.419,A -85,B 0,C 180,E1 -22947.669,E2 -22947.669} C_VEL
LIN {X 0,Y 174.063,Z 680.95,A -85,B 0,C 180,E1 -22952.315,E2 -22952.315} C_VEL
LIN {X 0,Y 175.879,Z 676.298,A -85,B 0,C 180,E1 -22956.886,E2 -22956.886} C_VEL
LIN {X 0,Y 178.594,Z 670.277,A -85,B 0,C 180,E1 -22961.348,E2 -22961.348} C_VEL
LIN {X 0,Y 182.02,Z 662.733,A -85,B 0,C 180,E1 -22965.681,E2 -22965.681} C_VEL
LIN {X 0,Y 185.65,Z 654.704,A -85,B 0,C 180,E1 -22969.344,E2 -22969.344} C_VEL
LIN {X 0,Y 189.842,Z 645.045,A -85,B 0,C 180,E1 -22972.875,E2 -22972.875} C_VEL
LIN {X 0,Y 194.47,Z 633.365,A -85,B 0,C 180,E1 -22976.277,E2 -22976.277} C_VEL
LIN {X 0,Y 198.3,Z 622.425,A -85,B 0,C 180,E1 -22978.874,E2 -22978.874} C_VEL
LIN {X 0,Y 202.149,Z 610.492,A -85,B 0,C 180,E1 -22981.141,E2 -22981.141} C_VEL
LIN {X 0,Y 205.725,Z 597.536,A -85,B 0,C 180,E1 -22983.134,E2 -22983.134} C_VEL
LIN {X 0,Y 208.999,Z 583.249,A -85,B 0,C 180,E1 -22984.866,E2 -22984.866} C_VEL
LIN {X 0,Y 211.712,Z 568.214,A -85,B 0,C 180,E1 -22986.249,E2 -22986.249} C_VEL
LIN {X 0,Y 213.733,Z 552.747,A -85,B 0,C 180,E1 -22987.274,E2 -22987.274} C_VEL
LIN {X 0,Y 214.789,Z 537.197,A -85,B 0,C 180,E1 -22987.993,E2 -22987.993} C_VEL
LIN {X 0,Y 217.451,Z 489.116,A -85,B 0,C 180,E1 -22989.509,E2 -22989.509} C_VEL
LIN {X 0,Y 217.956,Z 479.102,A -85,B 0,C 180,E1 -22989.838,E2 -22989.838} C_VEL
LIN {X 0,Y 211.425,Z 466.105,A -85,B 0,C 180,E1 -22992.343,E2 -22992.343} C_VEL
LIN {X 0,Y 204.757,Z 454.502,A -85,B 0,C 180,E1 -22995.121,E2 -22995.121} C_VEL
LIN {X 0,Y 197.604,Z 443.605,A -85,B 0,C 180,E1 -22998.429,E2 -22998.429} C_VEL
LIN {X 0,Y 193.855,Z 438.379,A -85,B 0,C 180,E1 -23000.345,E2 -23000.345} C_VEL
LIN {X 0,Y 191.502,Z 435.132,A -85,B 0,C 180,E1 -23001.636,E2 -23001.636} C_VEL
LIN {X 0,Y 188.234,Z 430.807,A -85,B 0,C 180,E1 -23003.551,E2 -23003.551} C_VEL
LIN {X 0,Y 185.525,Z 427.26,A -85,B 0,C 180,E1 -23005.275,E2 -23005.275} C_VEL
LIN {X 0,Y 184.566,Z 426.083,A -85,B 0,C 180,E1 -23005.914,E2 -23005.914} C_VEL
LIN {X 0,Y 182.032,Z 423.267,A -85,B 0,C 180,E1 -23007.678,E2 -23007.678} C_VEL
LIN {X 0,Y 180.826,Z 421.185,A -85,B 0,C 180,E1 -23008.643,E2 -23008.643} C_VEL
LIN {X 0,Y 178.204,Z 419.015,A -85,B 0,C 180,E1 -23010.681,E2 -23010.681} C_VEL
LIN {X 0,Y 176.415,Z 415.681,A -85,B 0,C 180,E1 -23012.411,E2 -23012.411} C_VEL
LIN {X 0,Y 173.678,Z 414.065,A -85,B 0,C 180,E1 -23014.984,E2 -23014.984} C_VEL
LIN {X 0,Y 172.028,Z 411.845,A -85,B 0,C 180,E1 -23016.924,E2 -23016.924} C_VEL
LIN {X 0,Y 171.422,Z 409.755,A -85,B 0,C 180,E1 -23018.03,E2 -23018.03} C_VEL
LIN {X 0,Y 171.506,Z 409.73,A -85,B 0,C 180,E1 -23020.863,E2 -23020.863} C_VEL
LIN {X 0,Y 171.553,Z 409.705,A -85,B 0,C 180,E1 -23025.77,E2 -23025.77} C_VEL
LIN {X 0,Y 171.838,Z 409.637,A -85,B 0,C 180,E1 -23030.584,E2 -23030.584} C_VEL
LIN {X 0,Y 171.762,Z 409.712,A -85,B 0,C 180,E1 -23035.305,E2 -23035.305} C_VEL
LIN {X 0,Y 172.3,Z 409.639,A -85,B 0,C 180,E1 -23039.999,E2 -23039.999} C_VEL
LIN {X 0,Y 171.776,Z 409.693,A -85,B 0,C 180,E1 -23044.693,E2 -23044.693} C_VEL
LIN {X 0,Y 171.839,Z 409.686,A -85,B 0,C 180,E1 -23049.415,E2 -23049.415} C_VEL
LIN {X 0,Y 171.744,Z 409.857,A -85,B 0,C 180,E1 -23051.418,E2 -23051.418} C_VEL
LIN {X 0,Y 172.287,Z 411.947,A -85,B 0,C 180,E1 -23052.291,E2 -23052.291} C_VEL
LIN {X 0,Y 174.024,Z 414.278,A -85,B 0,C 180,E1 -23054.291,E2 -23054.291} C_VEL
LIN {X 0,Y 176.616,Z 415.858,A -85,B 0,C 180,E1 -23056.693,E2 -23056.693} C_VEL
LIN {X 0,Y 178.07,Z 418.717,A -85,B 0,C 180,E1 -23058.107,E2 -23058.107} C_VEL
LIN {X 0,Y 179.711,Z 420.994,A -85,B 0,C 180,E1 -23059.501,E2 -23059.501} C_VEL
LIN {X 0,Y 182.898,Z 425.461,A -85,B 0,C 180,E1 -23061.965,E2 -23061.965} C_VEL
LIN {X 0,Y 186.365,Z 430.97,A -85,B 0,C 180,E1 -23064.396,E2 -23064.396} C_VEL
LIN {X 0,Y 192.206,Z 440.801,A -85,B 0,C 180,E1 -23067.991,E2 -23067.991} C_VEL
LIN {X 0,Y 195.747,Z 447.262,A -85,B 0,C 180,E1 -23069.952,E2 -23069.952} C_VEL
LIN {X 0,Y 200.622,Z 456.725,A -85,B 0,C 180,E1 -23072.439,E2 -23072.439} C_VEL
LIN {X 0,Y 206.266,Z 469.155,A -85,B 0,C 180,E1 -23075.097,E2 -23075.097} C_VEL
LIN {X 0,Y 210.821,Z 480.264,A -85,B 0,C 180,E1 -23077.097,E2 -23077.097} C_VEL
LIN {X 0,Y 213.539,Z 487.941,A -85,B 0,C 180,E1 -23078.269,E2 -23078.269} C_VEL
LIN {X 0,Y 215.708,Z 527.325,A -85,B 0,C 180,E1 -23080.706,E2 -23080.706} C_VEL
LIN {X 0,Y 211.906,Z 585.907,A -85,B 0,C 180,E1 -23082.442,E2 -23082.442} C_VEL
LIN {X 0,Y 210.834,Z 591.714,A -85,B 0,C 180,E1 -23082.528,E2 -23082.528} C_VEL
LIN {X 0,Y 207.512,Z 601.061,A -85,B 0,C 180,E1 -23082.461,E2 -23082.461} C_VEL
LIN {X 0,Y 203.839,Z 610.279,A -85,B 0,C 180,E1 -23082.494,E2 -23082.494} C_VEL
LIN {X 0,Y 202.277,Z 615.884,A -85,B 0,C 180,E1 -23082.797,E2 -23082.797} C_VEL
LIN {X 0,Y 198.753,Z 630.48,A -85,B 0,C 180,E1 -23084.09,E2 -23084.09} C_VEL
LIN {X 0,Y 194.811,Z 643.911,A -85,B 0,C 180,E1 -23085.656,E2 -23085.656} C_VEL
LIN {X 0,Y 190.014,Z 657.651,A -85,B 0,C 180,E1 -23087.708,E2 -23087.708} C_VEL
LIN {X 0,Y 186.776,Z 665.999,A -85,B 0,C 180,E1 -23089.235,E2 -23089.235} C_VEL
LIN {X 0,Y 182.218,Z 677.673,A -85,B 0,C 180,E1 -23091.895,E2 -23091.895} C_VEL
LIN {X 0,Y 177.481,Z 688.553,A -85,B 0,C 180,E1 -23094.958,E2 -23094.958} C_VEL
LIN {X 0,Y 172.841,Z 699.273,A -85,B 0,C 180,E1 -23098.787,E2 -23098.787} C_VEL
LIN {X 0,Y 169.12,Z 708.166,A -85,B 0,C 180,E1 -23102.798,E2 -23102.798} C_VEL
LIN {X 0,Y 166.706,Z 714.675,A -85,B 0,C 180,E1 -23106.39,E2 -23106.39} C_VEL
LIN {X 0,Y 164.442,Z 721.818,A -85,B 0,C 180,E1 -23111.304,E2 -23111.304} C_VEL
LIN {X 0,Y 163.42,Z 727.475,A -85,B 0,C 180,E1 -23116.318,E2 -23116.318} C_VEL
LIN {X 0,Y 163.51,Z 731.734,A -85,B 0,C 180,E1 -23121.333,E2 -23121.333} C_VEL
LIN {X 0,Y 163.993,Z 734.019,A -85,B 0,C 180,E1 -23125.082,E2 -23125.082} C_VEL
LIN {X 0,Y 165.032,Z 735.95,A -85,B 0,C 180,E1 -23129.999,E2 -23129.999} C_VEL
LIN {X 0,Y 163.876,Z 736.208,A -85,B 0,C 180,E1 -23134.919,E2 -23134.919} C_VEL
LIN {X 0,Y 163.132,Z 735.205,A -85,B 0,C 180,E1 -23139.922,E2 -23139.922} C_VEL
LIN {X 0,Y 163.329,Z 733.063,A -85,B 0,C 180,E1 -23144.961,E2 -23144.961} C_VEL
LIN {X 0,Y 165.066,Z 729.349,A -85,B 0,C 180,E1 -23150.498,E2 -23150.498} C_VEL
LIN {X 0,Y 168.36,Z 724,A -85,B 0,C 180,E1 -23155.994,E2 -23155.994} C_VEL
LIN {X 0,Y 172.609,Z 717.909,A -85,B 0,C 180,E1 -23160.592,E2 -23160.592} C_VEL
LIN {X 0,Y 178.026,Z 710.369,A -85,B 0,C 180,E1 -23164.917,E2 -23164.917} C_VEL
LIN {X 0,Y 183.665,Z 702.441,A -85,B 0,C 180,E1 -23168.446,E2 -23168.446} C_VEL
LIN {X 0,Y 190.16,Z 693.036,A -85,B 0,C 180,E1 -23171.699,E2 -23171.699} C_VEL
LIN {X 0,Y 196.461,Z 683.168,A -85,B 0,C 180,E1 -23174.38,E2 -23174.38} C_VEL
LIN {X 0,Y 203.374,Z 671.353,A -85,B 0,C 180,E1 -23176.885,E2 -23176.885} C_VEL
LIN {X 0,Y 209.889,Z 659.025,A -85,B 0,C 180,E1 -23178.883,E2 -23178.883} C_VEL
LIN {X 0,Y 216.131,Z 645.542,A -85,B 0,C 180,E1 -23180.557,E2 -23180.557} C_VEL
LIN {X 0,Y 221.213,Z 632.369,A -85,B 0,C 180,E1 -23181.839,E2 -23181.839} C_VEL
LIN {X 0,Y 225.823,Z 618.053,A -85,B 0,C 180,E1 -23182.888,E2 -23182.888} C_VEL
LIN {X 0,Y 229.428,Z 603.403,A -85,B 0,C 180,E1 -23183.706,E2 -23183.706} C_VEL
LIN {X 0,Y 231.949,Z 588.57,A -85,B 0,C 180,E1 -23184.329,E2 -23184.329} C_VEL
LIN {X 0,Y 233.93,Z 568.329,A -85,B 0,C 180,E1 -23184.9,E2 -23184.9} C_VEL
LIN {X 0,Y 236.817,Z 531.592,A -85,B 0,C 180,E1 -23185.863,E2 -23185.863} C_VEL
LIN {X 0,Y 236.254,Z 514.768,A -85,B 0,C 180,E1 -23187.086,E2 -23187.086} C_VEL
LIN {X 0,Y 232.037,Z 503.293,A -85,B 0,C 180,E1 -23189.712,E2 -23189.712} C_VEL
LIN {X 0,Y 227.971,Z 493.343,A -85,B 0,C 180,E1 -23192.518,E2 -23192.518} C_VEL
LIN {X 0,Y 224.894,Z 486.321,A -85,B 0,C 180,E1 -23194.904,E2 -23194.904} C_VEL
LIN {X 0,Y 222.82,Z 481.777,A -85,B 0,C 180,E1 -23196.689,E2 -23196.689} C_VEL
LIN {X 0,Y 220.089,Z 475.937,A -85,B 0,C 180,E1 -23199.356,E2 -23199.356} C_VEL
LIN {X 0,Y 216.941,Z 469.128,A -85,B 0,C 180,E1 -23203.17,E2 -23203.17} C_VEL
LIN {X 0,Y 213.806,Z 462.187,A -85,B 0,C 180,E1 -23208.846,E2 -23208.846} C_VEL
LIN {X 0,Y 212.924,Z 459.59,A -85,B 0,C 180,E1 -23211.805,E2 -23211.805} C_VEL
LIN {X 0,Y 212.653,Z 459.336,A -85,B 0,C 180,E1 -23220,E2 -23220} C_VEL
LIN {X 0,Y 213.102,Z 459.824,A -85,B 0,C 180,E1 -23221.772,E2 -23221.772} C_VEL
LIN {X 0,Y 215.067,Z 463.59,A -85,B 0,C 180,E1 -23226.565,E2 -23226.565} C_VEL
LIN {X 0,Y 216.209,Z 464.778,A -85,B 0,C 180,E1 -23228.323,E2 -23228.323} C_VEL
LIN {X 0,Y 218.583,Z 468.602,A -85,B 0,C 180,E1 -23231.451,E2 -23231.451} C_VEL
LIN {X 0,Y 219.585,Z 469.954,A -85,B 0,C 180,E1 -23232.543,E2 -23232.543} C_VEL
LIN {X 0,Y 222.597,Z 474.521,A -85,B 0,C 180,E1 -23235.458,E2 -23235.458} C_VEL
LIN {X 0,Y 225.933,Z 479.609,A -85,B 0,C 180,E1 -23238.183,E2 -23238.183} C_VEL
LIN {X 0,Y 230.178,Z 486.459,A -85,B 0,C 180,E1 -23241.171,E2 -23241.171} C_VEL
LIN {X 0,Y 235.165,Z 495.019,A -85,B 0,C 180,E1 -23244.208,E2 -23244.208} C_VEL
LIN {X 0,Y 239.008,Z 502.347,A -85,B 0,C 180,E1 -23246.321,E2 -23246.321} C_VEL
LIN {X 0,Y 235.851,Z 546.189,A -85,B 0,C 180,E1 -23247.642,E2 -23247.642} C_VEL
LIN {X 0,Y 234.079,Z 561.433,A -85,B 0,C 180,E1 -23248.369,E2 -23248.369} C_VEL
LIN {X 0,Y 231.854,Z 573.859,A -85,B 0,C 180,E1 -23249.164,E2 -23249.164} C_VEL
LIN {X 0,Y 228.657,Z 587.307,A -85,B 0,C 180,E1 -23250.267,E2 -23250.267} C_VEL
LIN {X 0,Y 224.902,Z 600.082,A -85,B 0,C 180,E1 -23251.624,E2 -23251.624} C_VEL
LIN {X 0,Y 219.879,Z 613.545,A -85,B 0,C 180,E1 -23253.359,E2 -23253.359} C_VEL
LIN {X 0,Y 214.418,Z 625.91,A -85,B 0,C 180,E1 -23255.383,E2 -23255.383} C_VEL
LIN {X 0,Y 208.278,Z 637.871,A -85,B 0,C 180,E1 -23257.868,E2 -23257.868} C_VEL
LIN {X 0,Y 201.772,Z 648.841,A -85,B 0,C 180,E1 -23260.752,E2 -23260.752} C_VEL
LIN {X 0,Y 196.027,Z 657.46,A -85,B 0,C 180,E1 -23263.594,E2 -23263.594} C_VEL
LIN {X 0,Y 190.199,Z 665.324,A -85,B 0,C 180,E1 -23266.878,E2 -23266.878} C_VEL
LIN {X 0,Y 184.04,Z 672.86,A -85,B 0,C 180,E1 -23270.946,E2 -23270.946} C_VEL
LIN {X 0,Y 178.615,Z 678.89,A -85,B 0,C 180,E1 -23275.352,E2 -23275.352} C_VEL
LIN {X 0,Y 175.286,Z 682.203,A -85,B 0,C 180,E1 -23278.587,E2 -23278.587} C_VEL
LIN {X 0,Y 171.497,Z 685.687,A -85,B 0,C 180,E1 -23283.208,E2 -23283.208} C_VEL
LIN {X 0,Y 168.593,Z 687.955,A -85,B 0,C 180,E1 -23287.966,E2 -23287.966} C_VEL
LIN {X 0,Y 166.654,Z 689.032,A -85,B 0,C 180,E1 -23292.832,E2 -23292.832} C_VEL
LIN {X 0,Y 165.614,Z 688.958,A -85,B 0,C 180,E1 -23297.751,E2 -23297.751} C_VEL
LIN {X 0,Y 165.226,Z 687.816,A -85,B 0,C 180,E1 -23302.67,E2 -23302.67} C_VEL
LIN {X 0,Y 165.699,Z 685.562,A -85,B 0,C 180,E1 -23307.57,E2 -23307.57} C_VEL
LIN {X 0,Y 167.033,Z 682.148,A -85,B 0,C 180,E1 -23312.412,E2 -23312.412} C_VEL
LIN {X 0,Y 168.909,Z 677.556,A -85,B 0,C 180,E1 -23317.171,E2 -23317.171} C_VEL
LIN {X 0,Y 171.745,Z 671.589,A -85,B 0,C 180,E1 -23321.807,E2 -23321.807} C_VEL
LIN {X 0,Y 175.32,Z 664.118,A -85,B 0,C 180,E1 -23326.297,E2 -23326.297} C_VEL
LIN {X 0,Y 179.068,Z 656.141,A -85,B 0,C 180,E1 -23330.086,E2 -23330.086} C_VEL
LIN {X 0,Y 183.438,Z 646.565,A -85,B 0,C 180,E1 -23333.721,E2 -23333.721} C_VEL
LIN {X 0,Y 187.552,Z 636.782,A -85,B 0,C 180,E1 -23336.723,E2 -23336.723} C_VEL
LIN {X 0,Y 191.9,Z 625.201,A -85,B 0,C 180,E1 -23339.631,E2 -23339.631} C_VEL
LIN {X 0,Y 195.799,Z 613.648,A -85,B 0,C 180,E1 -23341.967,E2 -23341.967} C_VEL
LIN {X 0,Y 199.561,Z 601.154,A -85,B 0,C 180,E1 -23343.992,E2 -23343.992} C_VEL
LIN {X 0,Y 202.928,Z 587.552,A -85,B 0,C 180,E1 -23345.763,E2 -23345.763} C_VEL
LIN {X 0,Y 205.731,Z 573.539,A -85,B 0,C 180,E1 -23347.173,E2 -23347.173} C_VEL
LIN {X 0,Y 207.96,Z 558.564,A -85,B 0,C 180,E1 -23348.298,E2 -23348.298} C_VEL
LIN {X 0,Y 209.361,Z 544.256,A -85,B 0,C 180,E1 -23349.056,E2 -23349.056} C_VEL
LIN {X 0,Y 211.536,Z 504.868,A -85,B 0,C 180,E1 -23350.398,E2 -23350.398} C_VEL
LIN {X 0,Y 213.019,Z 481.881,A -85,B 0,C 180,E1 -23351.089,E2 -23351.089} C_VEL
LIN {X 0,Y 206.641,Z 469.208,A -85,B 0,C 180,E1 -23353.693,E2 -23353.693} C_VEL
LIN {X 0,Y 200.456,Z 458.403,A -85,B 0,C 180,E1 -23356.444,E2 -23356.444} C_VEL
LIN {X 0,Y 193.799,Z 448.167,A -85,B 0,C 180,E1 -23359.732,E2 -23359.732} C_VEL
LIN {X 0,Y 189.221,Z 441.504,A -85,B 0,C 180,E1 -23362.284,E2 -23362.284} C_VEL
LIN {X 0,Y 185.748,Z 436.892,A -85,B 0,C 180,E1 -23364.403,E2 -23364.403} C_VEL
LIN {X 0,Y 182.438,Z 432.486,A -85,B 0,C 180,E1 -23366.641,E2 -23366.641} C_VEL
LIN {X 0,Y 179.708,Z 429.222,A -85,B 0,C 180,E1 -23368.655,E2 -23368.655} C_VEL
LIN {X 0,Y 178.661,Z 427.615,A -85,B 0,C 180,E1 -23369.519,E2 -23369.519} C_VEL
LIN {X 0,Y 176.074,Z 425.06,A -85,B 0,C 180,E1 -23371.685,E2 -23371.685} C_VEL
LIN {X 0,Y 174.545,Z 422.396,A -85,B 0,C 180,E1 -23373.226,E2 -23373.226} C_VEL
LIN {X 0,Y 171.678,Z 420.259,A -85,B 0,C 180,E1 -23376.155,E2 -23376.155} C_VEL
LIN {X 0,Y 170.063,Z 417.383,A -85,B 0,C 180,E1 -23378.324,E2 -23378.324} C_VEL
LIN {X 0,Y 169.786,Z 416.664,A -85,B 0,C 180,E1 -23378.764,E2 -23378.764} C_VEL
LIN {X 0,Y 166.454,Z 414.731,A -85,B 0,C 180,E1 -23384.071,E2 -23384.071} C_VEL
LIN {X 0,Y 165.019,Z 412.112,A -85,B 0,C 180,E1 -23388.293,E2 -23388.293} C_VEL
LIN {X 0,Y 164.775,Z 410.512,A -85,B 0,C 180,E1 -23390.176,E2 -23390.176} C_VEL
LIN {X 0,Y 164.812,Z 410.541,A -85,B 0,C 180,E1 -23392.649,E2 -23392.649} C_VEL
LIN {X 0,Y 165.263,Z 410.514,A -85,B 0,C 180,E1 -23399.999,E2 -23399.999} C_VEL
LIN {X 0,Y 165.204,Z 410.713,A -85,B 0,C 180,E1 -23400.685,E2 -23400.685} C_VEL
LIN {X 0,Y 165.774,Z 413.169,A -85,B 0,C 180,E1 -23403.037,E2 -23403.037} C_VEL
LIN {X 0,Y 167.244,Z 415.144,A -85,B 0,C 180,E1 -23406.333,E2 -23406.333} C_VEL
LIN {X 0,Y 170.099,Z 416.738,A -85,B 0,C 180,E1 -23410.547,E2 -23410.547} C_VEL
LIN {X 0,Y 171.302,Z 419.541,A -85,B 0,C 180,E1 -23412.288,E2 -23412.288} C_VEL
LIN {X 0,Y 173.582,Z 421.832,A -85,B 0,C 180,E1 -23414.79,E2 -23414.79} C_VEL
LIN {X 0,Y 174.832,Z 422.655,A -85,B 0,C 180,E1 -23415.97,E2 -23415.97} C_VEL
LIN {X 0,Y 176.769,Z 425.871,A -85,B 0,C 180,E1 -23417.852,E2 -23417.852} C_VEL
LIN {X 0,Y 180.65,Z 431.615,A -85,B 0,C 180,E1 -23421.091,E2 -23421.091} C_VEL
LIN {X 0,Y 183.819,Z 436.862,A -85,B 0,C 180,E1 -23423.444,E2 -23423.444} C_VEL
LIN {X 0,Y 189.344,Z 446.498,A -85,B 0,C 180,E1 -23427.045,E2 -23427.045} C_VEL
LIN {X 0,Y 192.754,Z 452.933,A -85,B 0,C 180,E1 -23429.037,E2 -23429.037} C_VEL
LIN {X 0,Y 197.438,Z 462.464,A -85,B 0,C 180,E1 -23431.565,E2 -23431.565} C_VEL
LIN {X 0,Y 202.363,Z 473.683,A -85,B 0,C 180,E1 -23434.023,E2 -23434.023} C_VEL
LIN {X 0,Y 206.605,Z 484.341,A -85,B 0,C 180,E1 -23436.004,E2 -23436.004} C_VEL
LIN {X 0,Y 208.766,Z 490.592,A -85,B 0,C 180,E1 -23436.995,E2 -23436.995} C_VEL
LIN {X 0,Y 210.656,Z 527.936,A -85,B 0,C 180,E1 -23439.379,E2 -23439.379} C_VEL
LIN {X 0,Y 206.515,Z 588.2,A -85,B 0,C 180,E1 -23441.195,E2 -23441.195} C_VEL
LIN {X 0,Y 204.457,Z 604.13,A -85,B 0,C 180,E1 -23441.984,E2 -23441.984} C_VEL
LIN {X 0,Y 202.277,Z 615.884,A -85,B 0,C 180,E1 -23442.797,E2 -23442.797} C_VEL
LIN {X 0,Y 200.531,Z 621.444,A -85,B 0,C 180,E1 -23443.119,E2 -23443.119} C_VEL
LIN {X 0,Y 196.004,Z 630.22,A -85,B 0,C 180,E1 -23443.409,E2 -23443.409} C_VEL
LIN {X 0,Y 191.233,Z 638.856,A -85,B 0,C 180,E1 -23443.848,E2 -23443.848} C_VEL
LIN {X 0,Y 189.085,Z 643.986,A -85,B 0,C 180,E1 -23444.409,E2 -23444.409} C_VEL
LIN {X 0,Y 184.21,Z 657.335,A -85,B 0,C 180,E1 -23446.459,E2 -23446.459} C_VEL
LIN {X 0,Y 180.841,Z 665.655,A -85,B 0,C 180,E1 -23448.017,E2 -23448.017} C_VEL
LIN {X 0,Y 175.733,Z 678.09,A -85,B 0,C 180,E1 -23450.959,E2 -23450.959} C_VEL
LIN {X 0,Y 170.863,Z 688.737,A -85,B 0,C 180,E1 -23454.117,E2 -23454.117} C_VEL
LIN {X 0,Y 166.316,Z 698.677,A -85,B 0,C 180,E1 -23457.837,E2 -23457.837} C_VEL
LIN {X 0,Y 162.232,Z 707.983,A -85,B 0,C 180,E1 -23462.244,E2 -23462.244} C_VEL
LIN {X 0,Y 159.358,Z 715.292,A -85,B 0,C 180,E1 -23466.614,E2 -23466.614} C_VEL
LIN {X 0,Y 157.207,Z 722.104,A -85,B 0,C 180,E1 -23471.763,E2 -23471.763} C_VEL
LIN {X 0,Y 156.307,Z 727.446,A -85,B 0,C 180,E1 -23477.007,E2 -23477.007} C_VEL
LIN {X 0,Y 156.524,Z 731.428,A -85,B 0,C 180,E1 -23482.258,E2 -23482.258} C_VEL
LIN {X 0,Y 156.882,Z 732.912,A -85,B 0,C 180,E1 -23484.859,E2 -23484.859} C_VEL
LIN {X 0,Y 157.98,Z 734.899,A -85,B 0,C 180,E1 -23489.999,E2 -23489.999} C_VEL
LIN {X 0,Y 156.796,Z 735.17,A -85,B 0,C 180,E1 -23495.142,E2 -23495.142} C_VEL
LIN {X 0,Y 156.056,Z 734.199,A -85,B 0,C 180,E1 -23500.377,E2 -23500.377} C_VEL
LIN {X 0,Y 156.375,Z 732.099,A -85,B 0,C 180,E1 -23505.643,E2 -23505.643} C_VEL
LIN {X 0,Y 158.186,Z 728.682,A -85,B 0,C 180,E1 -23511.094,E2 -23511.094} C_VEL
LIN {X 0,Y 160.956,Z 724.468,A -85,B 0,C 180,E1 -23515.888,E2 -23515.888} C_VEL
LIN {X 0,Y 165.18,Z 718.745,A -85,B 0,C 180,E1 -23520.7,E2 -23520.7} C_VEL
LIN {X 0,Y 170.654,Z 711.634,A -85,B 0,C 180,E1 -23525.207,E2 -23525.207} C_VEL
LIN {X 0,Y 177.175,Z 702.943,A -85,B 0,C 180,E1 -23529.393,E2 -23529.393} C_VEL
LIN {X 0,Y 183.863,Z 693.813,A -85,B 0,C 180,E1 -23532.722,E2 -23532.722} C_VEL
LIN {X 0,Y 190.047,Z 684.649,A -85,B 0,C 180,E1 -23535.362,E2 -23535.362} C_VEL
LIN {X 0,Y 196.792,Z 673.837,A -85,B 0,C 180,E1 -23537.817,E2 -23537.817} C_VEL
LIN {X 0,Y 204.021,Z 661.026,A -85,B 0,C 180,E1 -23540.034,E2 -23540.034} C_VEL
LIN {X 0,Y 210.403,Z 648.193,A -85,B 0,C 180,E1 -23541.714,E2 -23541.714} C_VEL
LIN {X 0,Y 215.636,Z 635.885,A -85,B 0,C 180,E1 -23542.984,E2 -23542.984} C_VEL
LIN {X 0,Y 219.6,Z 624.739,A -85,B 0,C 180,E1 -23543.907,E2 -23543.907} C_VEL
LIN {X 0,Y 223.948,Z 609.761,A -85,B 0,C 180,E1 -23544.872,E2 -23544.872} C_VEL
LIN {X 0,Y 227.137,Z 595.006,A -85,B 0,C 180,E1 -23545.564,E2 -23545.564} C_VEL
LIN {X 0,Y 229.297,Z 579.342,A -85,B 0,C 180,E1 -23546.098,E2 -23546.098} C_VEL
LIN {X 0,Y 233.16,Z 532.473,A -85,B 0,C 180,E1 -23547.334,E2 -23547.334} C_VEL
LIN {X 0,Y 232.728,Z 518.226,A -85,B 0,C 180,E1 -23548.416,E2 -23548.416} C_VEL
LIN {X 0,Y 229.135,Z 508.05,A -85,B 0,C 180,E1 -23550.827,E2 -23550.827} C_VEL
LIN {X 0,Y 225.517,Z 498.763,A -85,B 0,C 180,E1 -23553.506,E2 -23553.506} C_VEL
LIN {X 0,Y 221.816,Z 489.765,A -85,B 0,C 180,E1 -23556.658,E2 -23556.658} C_VEL
LIN {X 0,Y 218.347,Z 482.069,A -85,B 0,C 180,E1 -23560.172,E2 -23560.172} C_VEL
LIN {X 0,Y 215.61,Z 475.798,A -85,B 0,C 180,E1 -23563.718,E2 -23563.718} C_VEL
LIN {X 0,Y 212.727,Z 468.95,A -85,B 0,C 180,E1 -23569.335,E2 -23569.335} C_VEL
LIN {X 0,Y 211.967,Z 466.585,A -85,B 0,C 180,E1 -23572.115,E2 -23572.115} C_VEL
LIN {X 0,Y 211.781,Z 466.382,A -85,B 0,C 180,E1 -23580,E2 -23580} C_VEL
LIN {X 0,Y 212.155,Z 466.84,A -85,B 0,C 180,E1 -23581.543,E2 -23581.543} C_VEL
LIN {X 0,Y 214.01,Z 470.529,A -85,B 0,C 180,E1 -23586.281,E2 -23586.281} C_VEL
LIN {X 0,Y 215.067,Z 471.737,A -85,B 0,C 180,E1 -23587.984,E2 -23587.984} C_VEL
LIN {X 0,Y 217.425,Z 475.537,A -85,B 0,C 180,E1 -23591.183,E2 -23591.183} C_VEL
LIN {X 0,Y 218.325,Z 476.921,A -85,B 0,C 180,E1 -23592.21,E2 -23592.21} C_VEL
LIN {X 0,Y 220.896,Z 480.943,A -85,B 0,C 180,E1 -23594.805,E2 -23594.805} C_VEL
LIN {X 0,Y 224.093,Z 486.042,A -85,B 0,C 180,E1 -23597.548,E2 -23597.548} C_VEL
LIN {X 0,Y 227.671,Z 491.957,A -85,B 0,C 180,E1 -23600.204,E2 -23600.204} C_VEL
LIN {X 0,Y 232.242,Z 500.082,A -85,B 0,C 180,E1 -23603.167,E2 -23603.167} C_VEL
LIN {X 0,Y 235.207,Z 505.786,A -85,B 0,C 180,E1 -23604.906,E2 -23604.906} C_VEL
LIN {X 0,Y 232.061,Z 548.326,A -85,B 0,C 180,E1 -23606.225,E2 -23606.225} C_VEL
LIN {X 0,Y 230.142,Z 563.487,A -85,B 0,C 180,E1 -23606.964,E2 -23606.964} C_VEL
LIN {X 0,Y 228.028,Z 574.745,A -85,B 0,C 180,E1 -23607.695,E2 -23607.695} C_VEL
LIN {X 0,Y 224.62,Z 588.573,A -85,B 0,C 180,E1 -23608.832,E2 -23608.832} C_VEL
LIN {X 0,Y 220.621,Z 601.607,A -85,B 0,C 180,E1 -23610.226,E2 -23610.226} C_VEL
LIN {X 0,Y 215.391,Z 615.049,A -85,B 0,C 180,E1 -23611.971,E2 -23611.971} C_VEL
LIN {X 0,Y 209.774,Z 627.269,A -85,B 0,C 180,E1 -23613.988,E2 -23613.988} C_VEL
LIN {X 0,Y 203.77,Z 638.554,A -85,B 0,C 180,E1 -23616.335,E2 -23616.335} C_VEL
LIN {X 0,Y 197.146,Z 649.36,A -85,B 0,C 180,E1 -23619.165,E2 -23619.165} C_VEL
LIN {X 0,Y 190.369,Z 659.057,A -85,B 0,C 180,E1 -23622.411,E2 -23622.411} C_VEL
LIN {X 0,Y 184.163,Z 667.049,A -85,B 0,C 180,E1 -23625.859,E2 -23625.859} C_VEL
LIN {X 0,Y 178.503,Z 673.582,A -85,B 0,C 180,E1 -23629.488,E2 -23629.488} C_VEL
LIN {X 0,Y 172.722,Z 679.683,A -85,B 0,C 180,E1 -23633.989,E2 -23633.989} C_VEL
LIN {X 0,Y 169.188,Z 683.053,A -85,B 0,C 180,E1 -23637.317,E2 -23637.317} C_VEL
LIN {X 0,Y 165.133,Z 686.592,A -85,B 0,C 180,E1 -23642.087,E2 -23642.087} C_VEL
LIN {X 0,Y 161.97,Z 688.912,A -85,B 0,C 180,E1 -23647.015,E2 -23647.015} C_VEL
LIN {X 0,Y 159.825,Z 690.021,A -85,B 0,C 180,E1 -23652.074,E2 -23652.074} C_VEL
LIN {X 0,Y 158.686,Z 689.994,A -85,B 0,C 180,E1 -23657.207,E2 -23657.207} C_VEL
LIN {X 0,Y 158.2,Z 688.906,A -85,B 0,C 180,E1 -23662.342,E2 -23662.342} C_VEL
LIN {X 0,Y 158.647,Z 686.705,A -85,B 0,C 180,E1 -23667.462,E2 -23667.462} C_VEL
LIN {X 0,Y 159.975,Z 683.351,A -85,B 0,C 180,E1 -23672.519,E2 -23672.519} C_VEL
LIN {X 0,Y 161.942,Z 678.802,A -85,B 0,C 180,E1 -23677.482,E2 -23677.482} C_VEL
LIN {X 0,Y 164.894,Z 672.884,A -85,B 0,C 180,E1 -23682.305,E2 -23682.305} C_VEL
LIN {X 0,Y 168.634,Z 665.484,A -85,B 0,C 180,E1 -23686.962,E2 -23686.962} C_VEL
LIN {X 0,Y 172.53,Z 657.57,A -85,B 0,C 180,E1 -23690.882,E2 -23690.882} C_VEL
LIN {X 0,Y 177.073,Z 648.081,A -85,B 0,C 180,E1 -23694.629,E2 -23694.629} C_VEL
LIN {X 0,Y 181.352,Z 638.398,A -85,B 0,C 180,E1 -23697.713,E2 -23697.713} C_VEL
LIN {X 0,Y 185.893,Z 626.932,A -85,B 0,C 180,E1 -23700.69,E2 -23700.69} C_VEL
LIN {X 0,Y 189.92,Z 615.537,A -85,B 0,C 180,E1 -23703.081,E2 -23703.081} C_VEL
LIN {X 0,Y 194.298,Z 601.687,A -85,B 0,C 180,E1 -23705.362,E2 -23705.362} C_VEL
LIN {X 0,Y 197.787,Z 587.97,A -85,B 0,C 180,E1 -23707.161,E2 -23707.161} C_VEL
LIN {X 0,Y 200.711,Z 573.776,A -85,B 0,C 180,E1 -23708.588,E2 -23708.588} C_VEL
LIN {X 0,Y 203.011,Z 558.675,A -85,B 0,C 180,E1 -23709.714,E2 -23709.714} C_VEL
LIN {X 0,Y 204.379,Z 544.903,A -85,B 0,C 180,E1 -23710.444,E2 -23710.444} C_VEL
LIN {X 0,Y 206.641,Z 505.915,A -85,B 0,C 180,E1 -23711.79,E2 -23711.79} C_VEL
LIN {X 0,Y 208.023,Z 484.425,A -85,B 0,C 180,E1 -23712.461,E2 -23712.461} C_VEL
LIN {X 0,Y 201.906,Z 472.163,A -85,B 0,C 180,E1 -23715.139,E2 -23715.139} C_VEL
LIN {X 0,Y 195.868,Z 461.691,A -85,B 0,C 180,E1 -23718.019,E2 -23718.019} C_VEL
LIN {X 0,Y 189.413,Z 451.474,A -85,B 0,C 180,E1 -23721.494,E2 -23721.494} C_VEL
LIN {X 0,Y 183.47,Z 443.145,A -85,B 0,C 180,E1 -23725.171,E2 -23725.171} C_VEL
LIN {X 0,Y 180.049,Z 438.576,A -85,B 0,C 180,E1 -23727.597,E2 -23727.597} C_VEL
LIN {X 0,Y 177.344,Z 434.999,A -85,B 0,C 180,E1 -23729.741,E2 -23729.741} C_VEL
LIN {X 0,Y 176.331,Z 433.832,A -85,B 0,C 180,E1 -23730.591,E2 -23730.591} C_VEL
LIN {X 0,Y 173.795,Z 430.811,A -85,B 0,C 180,E1 -23732.918,E2 -23732.918} C_VEL
LIN {X 0,Y 172.879,Z 429.145,A -85,B 0,C 180,E1 -23733.904,E2 -23733.904} C_VEL
LIN {X 0,Y 169.921,Z 426.579,A -85,B 0,C 180,E1 -23737.144,E2 -23737.144} C_VEL
LIN {X 0,Y 168.353,Z 423.557,A -85,B 0,C 180,E1 -23739.454,E2 -23739.454} C_VEL
LIN {X 0,Y 165.075,Z 421.279,A -85,B 0,C 180,E1 -23745.199,E2 -23745.199} C_VEL
LIN {X 0,Y 163.954,Z 418.642,A -85,B 0,C 180,E1 -23749.19,E2 -23749.19} C_VEL
LIN {X 0,Y 163.794,Z 417.539,A -85,B 0,C 180,E1 -23750.483,E2 -23750.483} C_VEL
LIN {X 0,Y 164.173,Z 417.756,A -85,B 0,C 180,E1 -23760.153,E2 -23760.153} C_VEL
LIN {X 0,Y 165.092,Z 420.874,A -85,B 0,C 180,E1 -23763.661,E2 -23763.661} C_VEL
LIN {X 0,Y 167.644,Z 423.056,A -85,B 0,C 180,E1 -23768.437,E2 -23768.437} C_VEL
LIN {X 0,Y 168.687,Z 423.736,A -85,B 0,C 180,E1 -23769.921,E2 -23769.921} C_VEL
LIN {X 0,Y 170.145,Z 426.632,A -85,B 0,C 180,E1 -23772.032,E2 -23772.032} C_VEL
LIN {X 0,Y 172.662,Z 428.951,A -85,B 0,C 180,E1 -23774.803,E2 -23774.803} C_VEL
LIN {X 0,Y 173.261,Z 429.664,A -85,B 0,C 180,E1 -23775.418,E2 -23775.418} C_VEL
LIN {X 0,Y 178.329,Z 437.546,A -85,B 0,C 180,E1 -23780.096,E2 -23780.096} C_VEL
LIN {X 0,Y 181.546,Z 443.059,A -85,B 0,C 180,E1 -23782.624,E2 -23782.624} C_VEL
LIN {X 0,Y 186.438,Z 452.051,A -85,B 0,C 180,E1 -23786.01,E2 -23786.01} C_VEL
LIN {X 0,Y 189.803,Z 458.659,A -85,B 0,C 180,E1 -23788.095,E2 -23788.095} C_VEL
LIN {X 0,Y 193.869,Z 467.217,A -85,B 0,C 180,E1 -23790.423,E2 -23790.423} C_VEL
LIN {X 0,Y 198.961,Z 479.215,A -85,B 0,C 180,E1 -23793.121,E2 -23793.121} C_VEL
LIN {X 0,Y 203.395,Z 490.976,A -85,B 0,C 180,E1 -23795.313,E2 -23795.313} C_VEL
LIN {X 0,Y 204.159,Z 493.844,A -85,B 0,C 180,E1 -23795.716,E2 -23795.716} C_VEL
LIN {X 0,Y 205.681,Z 528.104,A -85,B 0,C 180,E1 -23797.955,E2 -23797.955} C_VEL
LIN {X 0,Y 201.515,Z 587.277,A -85,B 0,C 180,E1 -23799.773,E2 -23799.773} C_VEL
LIN {X 0,Y 199.437,Z 602.904,A -85,B 0,C 180,E1 -23800.55,E2 -23800.55} C_VEL
LIN {X 0,Y 196.368,Z 618.435,A -85,B 0,C 180,E1 -23801.659,E2 -23801.659} C_VEL
LIN {X 0,Y 192.487,Z 633.293,A -85,B 0,C 180,E1 -23803.095,E2 -23803.095} C_VEL
LIN {X 0,Y 189.085,Z 643.986,A -85,B 0,C 180,E1 -23804.409,E2 -23804.409} C_VEL
LIN {X 0,Y 186.862,Z 649.076,A -85,B 0,C 180,E1 -23805.023,E2 -23805.023} C_VEL
LIN {X 0,Y 181.524,Z 657.026,A -85,B 0,C 180,E1 -23805.805,E2 -23805.805} C_VEL
LIN {X 0,Y 175.925,Z 664.702,A -85,B 0,C 180,E1 -23806.741,E2 -23806.741} C_VEL
LIN {X 0,Y 173.31,Z 669.246,A -85,B 0,C 180,E1 -23807.612,E2 -23807.612} C_VEL
LIN {X 0,Y 168.448,Z 680.27,A -85,B 0,C 180,E1 -23810.486,E2 -23810.486} C_VEL
LIN {X 0,Y 163.543,Z 690.457,A -85,B 0,C 180,E1 -23813.78,E2 -23813.78} C_VEL
LIN {X 0,Y 158.713,Z 700.481,A -85,B 0,C 180,E1 -23817.902,E2 -23817.902} C_VEL
LIN {X 0,Y 154.833,Z 708.875,A -85,B 0,C 180,E1 -23822.273,E2 -23822.273} C_VEL
LIN {X 0,Y 152.017,Z 715.899,A -85,B 0,C 180,E1 -23826.86,E2 -23826.86} C_VEL
LIN {X 0,Y 149.965,Z 722.382,A -85,B 0,C 180,E1 -23832.264,E2 -23832.264} C_VEL
LIN {X 0,Y 149.226,Z 727.415,A -85,B 0,C 180,E1 -23837.764,E2 -23837.764} C_VEL
LIN {X 0,Y 149.437,Z 730.294,A -85,B 0,C 180,E1 -23841.888,E2 -23841.888} C_VEL
LIN {X 0,Y 150.222,Z 732.978,A -85,B 0,C 180,E1 -23847.318,E2 -23847.318} C_VEL
LIN {X 0,Y 150.902,Z 733.839,A -85,B 0,C 180,E1 -23849.999,E2 -23849.999} C_VEL
LIN {X 0,Y 149.696,Z 734.129,A -85,B 0,C 180,E1 -23855.387,E2 -23855.387} C_VEL
LIN {X 0,Y 148.982,Z 733.192,A -85,B 0,C 180,E1 -23860.875,E2 -23860.875} C_VEL
LIN {X 0,Y 149.446,Z 731.135,A -85,B 0,C 180,E1 -23866.388,E2 -23866.388} C_VEL
LIN {X 0,Y 151.346,Z 727.968,A -85,B 0,C 180,E1 -23871.806,E2 -23871.806} C_VEL
LIN {X 0,Y 154.509,Z 723.576,A -85,B 0,C 180,E1 -23877.054,E2 -23877.054} C_VEL
LIN {X 0,Y 159.02,Z 717.902,A -85,B 0,C 180,E1 -23882.027,E2 -23882.027} C_VEL
LIN {X 0,Y 164.801,Z 710.847,A -85,B 0,C 180,E1 -23886.655,E2 -23886.655} C_VEL
LIN {X 0,Y 170.752,Z 703.379,A -85,B 0,C 180,E1 -23890.408,E2 -23890.408} C_VEL
LIN {X 0,Y 177.64,Z 694.551,A -85,B 0,C 180,E1 -23893.814,E2 -23893.814} C_VEL
LIN {X 0,Y 184.508,Z 684.941,A -85,B 0,C 180,E1 -23896.716,E2 -23896.716} C_VEL
LIN {X 0,Y 192.082,Z 673.358,A -85,B 0,C 180,E1 -23899.392,E2 -23899.392} C_VEL
LIN {X 0,Y 198.889,Z 661.845,A -85,B 0,C 180,E1 -23901.424,E2 -23901.424} C_VEL
LIN {X 0,Y 205.408,Z 649.397,A -85,B 0,C 180,E1 -23903.105,E2 -23903.105} C_VEL
LIN {X 0,Y 211.439,Z 635.834,A -85,B 0,C 180,E1 -23904.52,E2 -23904.52} C_VEL
LIN {X 0,Y 215.502,Z 624.843,A -85,B 0,C 180,E1 -23905.429,E2 -23905.429} C_VEL
LIN {X 0,Y 219.949,Z 610.223,A -85,B 0,C 180,E1 -23906.381,E2 -23906.381} C_VEL
LIN {X 0,Y 223.551,Z 594.268,A -85,B 0,C 180,E1 -23907.135,E2 -23907.135} C_VEL
LIN {X 0,Y 225.798,Z 578.638,A -85,B 0,C 180,E1 -23907.662,E2 -23907.662} C_VEL
LIN {X 0,Y 229.649,Z 533.633,A -85,B 0,C 180,E1 -23908.841,E2 -23908.841} C_VEL
LIN {X 0,Y 229.407,Z 521.791,A -85,B 0,C 180,E1 -23909.745,E2 -23909.745} C_VEL
LIN {X 0,Y 225.343,Z 509.998,A -85,B 0,C 180,E1 -23912.73,E2 -23912.73} C_VEL
LIN {X 0,Y 221.747,Z 500.505,A -85,B 0,C 180,E1 -23915.731,E2 -23915.731} C_VEL
LIN {X 0,Y 219.05,Z 493.943,A -85,B 0,C 180,E1 -23918.312,E2 -23918.312} C_VEL
LIN {X 0,Y 216.515,Z 487.941,A -85,B 0,C 180,E1 -23921.159,E2 -23921.159} C_VEL
LIN {X 0,Y 214.292,Z 482.436,A -85,B 0,C 180,E1 -23924.287,E2 -23924.287} C_VEL
LIN {X 0,Y 211.675,Z 475.799,A -85,B 0,C 180,E1 -23929.78,E2 -23929.78} C_VEL
LIN {X 0,Y 211.033,Z 473.625,A -85,B 0,C 180,E1 -23932.345,E2 -23932.345} C_VEL
LIN {X 0,Y 210.912,Z 473.404,A -85,B 0,C 180,E1 -23940,E2 -23940} C_VEL
LIN {X 0,Y 211.21,Z 473.861,A -85,B 0,C 180,E1 -23941.311,E2 -23941.311} C_VEL
LIN {X 0,Y 213.136,Z 477.658,A -85,B 0,C 180,E1 -23946.307,E2 -23946.307} C_VEL
LIN {X 0,Y 213.95,Z 478.733,A -85,B 0,C 180,E1 -23947.669,E2 -23947.669} C_VEL
LIN {X 0,Y 216.274,Z 482.482,A -85,B 0,C 180,E1 -23950.918,E2 -23950.918} C_VEL
LIN {X 0,Y 219.369,Z 487.581,A -85,B 0,C 180,E1 -23954.281,E2 -23954.281} C_VEL
LIN {X 0,Y 223.364,Z 494.116,A -85,B 0,C 180,E1 -23957.769,E2 -23957.769} C_VEL
LIN {X 0,Y 228.17,Z 502.785,A -85,B 0,C 180,E1 -23961.285,E2 -23961.285} C_VEL
LIN {X 0,Y 231.595,Z 509.556,A -85,B 0,C 180,E1 -23963.487,E2 -23963.487} C_VEL
LIN {X 0,Y 228.54,Z 548.958,A -85,B 0,C 180,E1 -23964.702,E2 -23964.702} C_VEL
LIN {X 0,Y 226.585,Z 564.047,A -85,B 0,C 180,E1 -23965.43,E2 -23965.43} C_VEL
LIN {X 0,Y 224.253,Z 576.069,A -85,B 0,C 180,E1 -23966.205,E2 -23966.205} C_VEL
LIN {X 0,Y 220.592,Z 590.237,A -85,B 0,C 180,E1 -23967.37,E2 -23967.37} C_VEL
LIN {X 0,Y 216.056,Z 604.232,A -85,B 0,C 180,E1 -23968.901,E2 -23968.901} C_VEL
LIN {X 0,Y 211.072,Z 616.486,A -85,B 0,C 180,E1 -23970.513,E2 -23970.513} C_VEL
LIN {X 0,Y 205.248,Z 628.63,A -85,B 0,C 180,E1 -23972.525,E2 -23972.525} C_VEL
LIN {X 0,Y 198.703,Z 640.375,A -85,B 0,C 180,E1 -23975.005,E2 -23975.005} C_VEL
LIN {X 0,Y 192.671,Z 649.857,A -85,B 0,C 180,E1 -23977.502,E2 -23977.502} C_VEL
LIN {X 0,Y 185.592,Z 659.659,A -85,B 0,C 180,E1 -23980.771,E2 -23980.771} C_VEL
LIN {X 0,Y 179.048,Z 667.712,A -85,B 0,C 180,E1 -23984.249,E2 -23984.249} C_VEL
LIN {X 0,Y 173.085,Z 674.305,A -85,B 0,C 180,E1 -23987.938,E2 -23987.938} C_VEL
LIN {X 0,Y 167.087,Z 680.336,A -85,B 0,C 180,E1 -23992.42,E2 -23992.42} C_VEL
LIN {X 0,Y 163.179,Z 683.905,A -85,B 0,C 180,E1 -23995.953,E2 -23995.953} C_VEL
LIN {X 0,Y 158.823,Z 687.501,A -85,B 0,C 180,E1 -24000.874,E2 -24000.874} C_VEL
LIN {X 0,Y 155.404,Z 689.853,A -85,B 0,C 180,E1 -24005.984,E2 -24005.984} C_VEL
LIN {X 0,Y 153.038,Z 691.01,A -85,B 0,C 180,E1 -24011.25,E2 -24011.25} C_VEL
LIN {X 0,Y 151.754,Z 691.033,A -85,B 0,C 180,E1 -24016.613,E2 -24016.613} C_VEL
LIN {X 0,Y 151.177,Z 689.997,A -85,B 0,C 180,E1 -24021.984,E2 -24021.984} C_VEL
LIN {X 0,Y 151.599,Z 687.847,A -85,B 0,C 180,E1 -24027.344,E2 -24027.344} C_VEL
LIN {X 0,Y 152.92,Z 684.548,A -85,B 0,C 180,E1 -24032.635,E2 -24032.635} C_VEL
LIN {X 0,Y 154.998,Z 680.026,A -85,B 0,C 180,E1 -24037.819,E2 -24037.819} C_VEL
LIN {X 0,Y 158.049,Z 674.169,A -85,B 0,C 180,E1 -24042.847,E2 -24042.847} C_VEL
LIN {X 0,Y 161.948,Z 666.836,A -85,B 0,C 180,E1 -24047.685,E2 -24047.685} C_VEL
LIN {X 0,Y 166.656,Z 657.791,A -85,B 0,C 180,E1 -24052.305,E2 -24052.305} C_VEL
LIN {X 0,Y 171.482,Z 648.139,A -85,B 0,C 180,E1 -24056.141,E2 -24056.141} C_VEL
LIN {X 0,Y 176.803,Z 636.469,A -85,B 0,C 180,E1 -24059.794,E2 -24059.794} C_VEL
LIN {X 0,Y 181.553,Z 624.429,A -85,B 0,C 180,E1 -24062.816,E2 -24062.816} C_VEL
LIN {X 0,Y 185.956,Z 612.327,A -85,B 0,C 180,E1 -24065.195,E2 -24065.195} C_VEL
LIN {X 0,Y 190.027,Z 599.127,A -85,B 0,C 180,E1 -24067.273,E2 -24067.273} C_VEL
LIN {X 0,Y 193.508,Z 585.467,A -85,B 0,C 180,E1 -24068.959,E2 -24068.959} C_VEL
LIN {X 0,Y 196.455,Z 570.544,A -85,B 0,C 180,E1 -24070.376,E2 -24070.376} C_VEL
LIN {X 0,Y 198.682,Z 555.091,A -85,B 0,C 180,E1 -24071.42,E2 -24071.42} C_VEL
LIN {X 0,Y 199.941,Z 538.756,A -85,B 0,C 180,E1 -24072.181,E2 -24072.181} C_VEL
LIN {X 0,Y 202.427,Z 499.272,A -85,B 0,C 180,E1 -24073.478,E2 -24073.478} C_VEL
LIN {X 0,Y 203.15,Z 487.095,A -85,B 0,C 180,E1 -24073.893,E2 -24073.893} C_VEL
LIN {X 0,Y 197.588,Z 475.774,A -85,B 0,C 180,E1 -24076.505,E2 -24076.505} C_VEL
LIN {X 0,Y 192.473,Z 466.78,A -85,B 0,C 180,E1 -24079.104,E2 -24079.104} C_VEL
LIN {X 0,Y 186.489,Z 457.083,A -85,B 0,C 180,E1 -24082.517,E2 -24082.517} C_VEL
LIN {X 0,Y 181.15,Z 449.323,A -85,B 0,C 180,E1 -24086.008,E2 -24086.008} C_VEL
LIN {X 0,Y 177.778,Z 444.729,A -85,B 0,C 180,E1 -24088.527,E2 -24088.527} C_VEL
LIN {X 0,Y 174.711,Z 440.52,A -85,B 0,C 180,E1 -24091.136,E2 -24091.136} C_VEL
LIN {X 0,Y 172.174,Z 437.496,A -85,B 0,C 180,E1 -24093.554,E2 -24093.554} C_VEL
LIN {X 0,Y 171.129,Z 435.763,A -85,B 0,C 180,E1 -24094.713,E2 -24094.713} C_VEL
LIN {X 0,Y 168.234,Z 432.895,A -85,B 0,C 180,E1 -24098.133,E2 -24098.133} C_VEL
LIN {X 0,Y 167.1,Z 430.552,A -85,B 0,C 180,E1 -24099.925,E2 -24099.925} C_VEL
LIN {X 0,Y 163.79,Z 427.843,A -85,B 0,C 180,E1 -24106.27,E2 -24106.27} C_VEL
LIN {X 0,Y 162.931,Z 425.22,A -85,B 0,C 180,E1 -24110.064,E2 -24110.064} C_VEL
LIN {X 0,Y 162.826,Z 424.564,A -85,B 0,C 180,E1 -24111.032,E2 -24111.032} C_VEL
LIN {X 0,Y 163.177,Z 424.79,A -85,B 0,C 180,E1 -24119.691,E2 -24119.691} C_VEL
LIN {X 0,Y 164.088,Z 427.881,A -85,B 0,C 180,E1 -24123.376,E2 -24123.376} C_VEL
LIN {X 0,Y 166.88,Z 430.166,A -85,B 0,C 180,E1 -24128.628,E2 -24128.628} C_VEL
LIN {X 0,Y 167.312,Z 430.642,A -85,B 0,C 180,E1 -24129.291,E2 -24129.291} C_VEL
LIN {X 0,Y 168.972,Z 433.704,A -85,B 0,C 180,E1 -24131.749,E2 -24131.749} C_VEL
LIN {X 0,Y 171.562,Z 436.266,A -85,B 0,C 180,E1 -24134.676,E2 -24134.676} C_VEL
LIN {X 0,Y 176.106,Z 443.639,A -85,B 0,C 180,E1 -24139.127,E2 -24139.127} C_VEL
LIN {X 0,Y 180.134,Z 450.922,A -85,B 0,C 180,E1 -24142.433,E2 -24142.433} C_VEL
LIN {X 0,Y 183.644,Z 457.634,A -85,B 0,C 180,E1 -24144.971,E2 -24144.971} C_VEL
LIN {X 0,Y 187.099,Z 464.752,A -85,B 0,C 180,E1 -24147.245,E2 -24147.245} C_VEL
LIN {X 0,Y 191.488,Z 474.578,A -85,B 0,C 180,E1 -24149.89,E2 -24149.89} C_VEL
LIN {X 0,Y 196.301,Z 486.54,A -85,B 0,C 180,E1 -24152.557,E2 -24152.557} C_VEL
LIN {X 0,Y 199.585,Z 495.983,A -85,B 0,C 180,E1 -24154.291,E2 -24154.291} C_VEL
LIN {X 0,Y 200.818,Z 529.952,A -85,B 0,C 180,E1 -24156.547,E2 -24156.547} C_VEL
LIN {X 0,Y 196.675,Z 586.169,A -85,B 0,C 180,E1 -24158.277,E2 -24158.277} C_VEL
LIN {X 0,Y 194.395,Z 602.44,A -85,B 0,C 180,E1 -24159.09,E2 -24159.09} C_VEL
LIN {X 0,Y 191.396,Z 617.265,A -85,B 0,C 180,E1 -24160.162,E2 -24160.162} C_VEL
LIN {X 0,Y 187.634,Z 631.208,A -85,B 0,C 180,E1 -24161.486,E2 -24161.486} C_VEL
LIN {X 0,Y 183.182,Z 644.888,A -85,B 0,C 180,E1 -24163.201,E2 -24163.201} C_VEL
LIN {X 0,Y 178.507,Z 657.001,A -85,B 0,C 180,E1 -24165.127,E2 -24165.127} C_VEL
LIN {X 0,Y 174.737,Z 665.946,A -85,B 0,C 180,E1 -24166.863,E2 -24166.863} C_VEL
LIN {X 0,Y 173.31,Z 669.246,A -85,B 0,C 180,E1 -24167.612,E2 -24167.612} C_VEL
LIN {X 0,Y 170.712,Z 673.737,A -85,B 0,C 180,E1 -24168.567,E2 -24168.567} C_VEL
LIN {X 0,Y 164.998,Z 680.664,A -85,B 0,C 180,E1 -24170.012,E2 -24170.012} C_VEL
LIN {X 0,Y 159.277,Z 687.249,A -85,B 0,C 180,E1 -24171.696,E2 -24171.696} C_VEL
LIN {X 0,Y 156.716,Z 691.066,A -85,B 0,C 180,E1 -24173.019,E2 -24173.019} C_VEL
LIN {X 0,Y 151.978,Z 700.377,A -85,B 0,C 180,E1 -24177.087,E2 -24177.087} C_VEL
LIN {X 0,Y 147.94,Z 708.607,A -85,B 0,C 180,E1 -24181.637,E2 -24181.637} C_VEL
LIN {X 0,Y 144.692,Z 716.352,A -85,B 0,C 180,E1 -24187.134,E2 -24187.134} C_VEL
LIN {X 0,Y 142.714,Z 722.513,A -85,B 0,C 180,E1 -24192.814,E2 -24192.814} C_VEL
LIN {X 0,Y 142.163,Z 727.278,A -85,B 0,C 180,E1 -24198.594,E2 -24198.594} C_VEL
LIN {X 0,Y 142.341,Z 729.158,A -85,B 0,C 180,E1 -24201.481,E2 -24201.481} C_VEL
LIN {X 0,Y 142.677,Z 730.697,A -85,B 0,C 180,E1 -24204.345,E2 -24204.345} C_VEL
LIN {X 0,Y 143.827,Z 732.769,A -85,B 0,C 180,E1 -24209.999,E2 -24209.999} C_VEL
LIN {X 0,Y 142.601,Z 733.087,A -85,B 0,C 180,E1 -24215.656,E2 -24215.656} C_VEL
LIN {X 0,Y 141.925,Z 732.185,A -85,B 0,C 180,E1 -24221.423,E2 -24221.423} C_VEL
LIN {X 0,Y 142.54,Z 730.17,A -85,B 0,C 180,E1 -24227.206,E2 -24227.206} C_VEL
LIN {X 0,Y 144.653,Z 727.043,A -85,B 0,C 180,E1 -24232.871,E2 -24232.871} C_VEL
LIN {X 0,Y 148.119,Z 722.683,A -85,B 0,C 180,E1 -24238.324,E2 -24238.324} C_VEL
LIN {X 0,Y 152.959,Z 717.062,A -85,B 0,C 180,E1 -24243.458,E2 -24243.458} C_VEL
LIN {X 0,Y 159.08,Z 710.062,A -85,B 0,C 180,E1 -24248.205,E2 -24248.205} C_VEL
LIN {X 0,Y 165.363,Z 702.658,A -85,B 0,C 180,E1 -24252.017,E2 -24252.017} C_VEL
LIN {X 0,Y 172.536,Z 693.898,A -85,B 0,C 180,E1 -24255.463,E2 -24255.463} C_VEL
LIN {X 0,Y 179.174,Z 685.101,A -85,B 0,C 180,E1 -24258.179,E2 -24258.179} C_VEL
LIN {X 0,Y 187.529,Z 672.883,A -85,B 0,C 180,E1 -24261.042,E2 -24261.042} C_VEL
LIN {X 0,Y 195.206,Z 660.306,A -85,B 0,C 180,E1 -24263.229,E2 -24263.229} C_VEL
LIN {X 0,Y 201.921,Z 647.769,A -85,B 0,C 180,E1 -24264.875,E2 -24264.875} C_VEL
LIN {X 0,Y 208.076,Z 634.088,A -85,B 0,C 180,E1 -24266.274,E2 -24266.274} C_VEL
LIN {X 0,Y 213.345,Z 619.974,A -85,B 0,C 180,E1 -24267.356,E2 -24267.356} C_VEL
LIN {X 0,Y 217.542,Z 605.516,A -85,B 0,C 180,E1 -24268.215,E2 -24268.215} C_VEL
LIN {X 0,Y 220.828,Z 589.908,A -85,B 0,C 180,E1 -24268.901,E2 -24268.901} C_VEL
LIN {X 0,Y 222.822,Z 574.663,A -85,B 0,C 180,E1 -24269.372,E2 -24269.372} C_VEL
LIN {X 0,Y 226.308,Z 535.163,A -85,B 0,C 180,E1 -24270.368,E2 -24270.368} C_VEL
LIN {X 0,Y 226.201,Z 525.481,A -85,B 0,C 180,E1 -24271.11,E2 -24271.11} C_VEL
LIN {X 0,Y 222.765,Z 515.024,A -85,B 0,C 180,E1 -24273.848,E2 -24273.848} C_VEL
LIN {X 0,Y 219.59,Z 506.133,A -85,B 0,C 180,E1 -24276.715,E2 -24276.715} C_VEL
LIN {X 0,Y 217.22,Z 500.047,A -85,B 0,C 180,E1 -24279.152,E2 -24279.152} C_VEL
LIN {X 0,Y 214.926,Z 494.192,A -85,B 0,C 180,E1 -24281.934,E2 -24281.934} C_VEL
LIN {X 0,Y 212.886,Z 488.905,A -85,B 0,C 180,E1 -24285.032,E2 -24285.032} C_VEL
LIN {X 0,Y 210.637,Z 482.629,A -85,B 0,C 180,E1 -24290.23,E2 -24290.23} C_VEL
LIN {X 0,Y 210.037,Z 480.636,A -85,B 0,C 180,E1 -24292.855,E2 -24292.855} C_VEL
LIN {X 0,Y 210.04,Z 480.453,A -85,B 0,C 180,E1 -24300,E2 -24300} C_VEL
LIN {X 0,Y 210.274,Z 480.981,A -85,B 0,C 180,E1 -24301.137,E2 -24301.137} C_VEL
LIN {X 0,Y 212.798,Z 485.604,A -85,B 0,C 180,E1 -24307.273,E2 -24307.273} C_VEL
LIN {X 0,Y 215.424,Z 490.133,A -85,B 0,C 180,E1 -24311.043,E2 -24311.043} C_VEL
LIN {X 0,Y 217.759,Z 494.094,A -85,B 0,C 180,E1 -24313.651,E2 -24313.651} C_VEL
LIN {X 0,Y 221.419,Z 500.263,A -85,B 0,C 180,E1 -24317.015,E2 -24317.015} C_VEL
LIN {X 0,Y 226.09,Z 509.08,A -85,B 0,C 180,E1 -24320.615,E2 -24320.615} C_VEL
LIN {X 0,Y 228.093,Z 513.097,A -85,B 0,C 180,E1 -24321.987,E2 -24321.987} C_VEL
LIN {X 0,Y 225.011,Z 551.569,A -85,B 0,C 180,E1 -24323.21,E2 -24323.21} C_VEL
LIN {X 0,Y 222.837,Z 567.052,A -85,B 0,C 180,E1 -24324.005,E2 -24324.005} C_VEL
LIN {X 0,Y 219.431,Z 582.429,A -85,B 0,C 180,E1 -24325.042,E2 -24325.042} C_VEL
LIN {X 0,Y 215.528,Z 595.921,A -85,B 0,C 180,E1 -24326.273,E2 -24326.273} C_VEL
LIN {X 0,Y 210.469,Z 609.773,A -85,B 0,C 180,E1 -24327.872,E2 -24327.872} C_VEL
LIN {X 0,Y 205.078,Z 621.807,A -85,B 0,C 180,E1 -24329.592,E2 -24329.592} C_VEL
LIN {X 0,Y 199.099,Z 633.193,A -85,B 0,C 180,E1 -24331.619,E2 -24331.619} C_VEL
LIN {X 0,Y 192.796,Z 643.696,A -85,B 0,C 180,E1 -24333.976,E2 -24333.976} C_VEL
LIN {X 0,Y 186.2,Z 653.337,A -85,B 0,C 180,E1 -24336.676,E2 -24336.676} C_VEL
LIN {X 0,Y 178.948,Z 662.69,A -85,B 0,C 180,E1 -24340.021,E2 -24340.021} C_VEL
LIN {X 0,Y 171.657,Z 671.001,A -85,B 0,C 180,E1 -24343.918,E2 -24343.918} C_VEL
LIN {X 0,Y 166.133,Z 676.714,A -85,B 0,C 180,E1 -24347.404,E2 -24347.404} C_VEL
LIN {X 0,Y 160.007,Z 682.433,A -85,B 0,C 180,E1 -24352.056,E2 -24352.056} C_VEL
LIN {X 0,Y 154.807,Z 686.743,A -85,B 0,C 180,E1 -24356.992,E2 -24356.992} C_VEL
LIN {X 0,Y 150.286,Z 689.962,A -85,B 0,C 180,E1 -24362.69,E2 -24362.69} C_VEL
LIN {X 0,Y 147.454,Z 691.535,A -85,B 0,C 180,E1 -24367.588,E2 -24367.588} C_VEL
LIN {X 0,Y 145.394,Z 692.18,A -85,B 0,C 180,E1 -24373.142,E2 -24373.142} C_VEL
LIN {X 0,Y 144.407,Z 691.711,A -85,B 0,C 180,E1 -24378.776,E2 -24378.776} C_VEL
LIN {X 0,Y 144.228,Z 690.177,A -85,B 0,C 180,E1 -24384.408,E2 -24384.408} C_VEL
LIN {X 0,Y 145.05,Z 687.518,A -85,B 0,C 180,E1 -24390.001,E2 -24390.001} C_VEL
LIN {X 0,Y 146.878,Z 683.636,A -85,B 0,C 180,E1 -24395.492,E2 -24395.492} C_VEL
LIN {X 0,Y 149.532,Z 678.52,A -85,B 0,C 180,E1 -24400.837,E2 -24400.837} C_VEL
LIN {X 0,Y 153.172,Z 672.011,A -85,B 0,C 180,E1 -24405.98,E2 -24405.98} C_VEL
LIN {X 0,Y 157.037,Z 665.021,A -85,B 0,C 180,E1 -24410.295,E2 -24410.295} C_VEL
LIN {X 0,Y 161.584,Z 656.632,A -85,B 0,C 180,E1 -24414.406,E2 -24414.406} C_VEL
LIN {X 0,Y 166.79,Z 646.541,A -85,B 0,C 180,E1 -24418.297,E2 -24418.297} C_VEL
LIN {X 0,Y 171.608,Z 636.239,A -85,B 0,C 180,E1 -24421.477,E2 -24421.477} C_VEL
LIN {X 0,Y 176.202,Z 625.081,A -85,B 0,C 180,E1 -24424.291,E2 -24424.291} C_VEL
LIN {X 0,Y 180.785,Z 612.909,A -85,B 0,C 180,E1 -24426.705,E2 -24426.705} C_VEL
LIN {X 0,Y 185.032,Z 599.611,A -85,B 0,C 180,E1 -24428.808,E2 -24428.808} C_VEL
LIN {X 0,Y 188.654,Z 585.84,A -85,B 0,C 180,E1 -24430.512,E2 -24430.512} C_VEL
LIN {X 0,Y 191.506,Z 571.906,A -85,B 0,C 180,E1 -24431.846,E2 -24431.846} C_VEL
LIN {X 0,Y 193.852,Z 556.592,A -85,B 0,C 180,E1 -24432.894,E2 -24432.894} C_VEL
LIN {X 0,Y 195.138,Z 541.288,A -85,B 0,C 180,E1 -24433.64,E2 -24433.64} C_VEL
LIN {X 0,Y 197.751,Z 500.939,A -85,B 0,C 180,E1 -24434.994,E2 -24434.994} C_VEL
LIN {X 0,Y 198.466,Z 489.848,A -85,B 0,C 180,E1 -24435.368,E2 -24435.368} C_VEL
LIN {X 0,Y 193.159,Z 479.052,A -85,B 0,C 180,E1 -24438.044,E2 -24438.044} C_VEL
LIN {X 0,Y 187.951,Z 469.735,A -85,B 0,C 180,E1 -24440.921,E2 -24440.921} C_VEL
LIN {X 0,Y 182.607,Z 461.129,A -85,B 0,C 180,E1 -24444.237,E2 -24444.237} C_VEL
LIN {X 0,Y 178.478,Z 454.987,A -85,B 0,C 180,E1 -24447.154,E2 -24447.154} C_VEL
LIN {X 0,Y 175.494,Z 450.754,A -85,B 0,C 180,E1 -24449.536,E2 -24449.536} C_VEL
LIN {X 0,Y 172.812,Z 446.988,A -85,B 0,C 180,E1 -24451.953,E2 -24451.953} C_VEL
LIN {X 0,Y 170.099,Z 443.373,A -85,B 0,C 180,E1 -24454.746,E2 -24454.746} C_VEL
LIN {X 0,Y 169.454,Z 442.399,A -85,B 0,C 180,E1 -24455.496,E2 -24455.496} C_VEL
LIN {X 0,Y 166.704,Z 439.366,A -85,B 0,C 180,E1 -24458.984,E2 -24458.984} C_VEL
LIN {X 0,Y 165.773,Z 437.404,A -85,B 0,C 180,E1 -24460.547,E2 -24460.547} C_VEL
LIN {X 0,Y 162.773,Z 434.773,A -85,B 0,C 180,E1 -24466.66,E2 -24466.66} C_VEL
LIN {X 0,Y 161.967,Z 432.119,A -85,B 0,C 180,E1 -24470.617,E2 -24470.617} C_VEL
LIN {X 0,Y 161.945,Z 431.767,A -85,B 0,C 180,E1 -24470.982,E2 -24470.982} C_VEL
LIN {X 0,Y 162.188,Z 431.703,A -85,B 0,C 180,E1 -24479.146,E2 -24479.146} C_VEL
LIN {X 0,Y 163.035,Z 434.788,A -85,B 0,C 180,E1 -24482.934,E2 -24482.934} C_VEL
LIN {X 0,Y 165.921,Z 437.349,A -85,B 0,C 180,E1 -24488.563,E2 -24488.563} C_VEL
LIN {X 0,Y 167.762,Z 440.684,A -85,B 0,C 180,E1 -24491.401,E2 -24491.401} C_VEL
LIN {X 0,Y 169.951,Z 442.943,A -85,B 0,C 180,E1 -24493.984,E2 -24493.984} C_VEL
LIN {X 0,Y 173.888,Z 449.585,A -85,B 0,C 180,E1 -24498.082,E2 -24498.082} C_VEL
LIN {X 0,Y 177.818,Z 457.049,A -85,B 0,C 180,E1 -24501.52,E2 -24501.52} C_VEL
LIN {X 0,Y 181.017,Z 463.491,A -85,B 0,C 180,E1 -24503.981,E2 -24503.981} C_VEL
LIN {X 0,Y 184.769,Z 471.544,A -85,B 0,C 180,E1 -24506.587,E2 -24506.587} C_VEL
LIN {X 0,Y 189.215,Z 482.234,A -85,B 0,C 180,E1 -24509.405,E2 -24509.405} C_VEL
LIN {X 0,Y 193.514,Z 493.842,A -85,B 0,C 180,E1 -24511.919,E2 -24511.919} C_VEL
LIN {X 0,Y 195.127,Z 498.843,A -85,B 0,C 180,E1 -24512.838,E2 -24512.838} C_VEL
LIN {X 0,Y 196.107,Z 530.79,A -85,B 0,C 180,E1 -24515.022,E2 -24515.022} C_VEL
LIN {X 0,Y 191.861,Z 585.984,A -85,B 0,C 180,E1 -24516.747,E2 -24516.747} C_VEL
LIN {X 0,Y 189.497,Z 601.958,A -85,B 0,C 180,E1 -24517.557,E2 -24517.557} C_VEL
LIN {X 0,Y 186.253,Z 617.221,A -85,B 0,C 180,E1 -24518.684,E2 -24518.684} C_VEL
LIN {X 0,Y 182.379,Z 630.992,A -85,B 0,C 180,E1 -24520.015,E2 -24520.015} C_VEL
LIN {X 0,Y 177.784,Z 644.544,A -85,B 0,C 180,E1 -24521.742,E2 -24521.742} C_VEL
LIN {X 0,Y 172.304,Z 658.092,A -85,B 0,C 180,E1 -24523.965,E2 -24523.965} C_VEL
LIN {X 0,Y 168.069,Z 667.593,A -85,B 0,C 180,E1 -24525.958,E2 -24525.958} C_VEL
LIN {X 0,Y 162.959,Z 678.725,A -85,B 0,C 180,E1 -24528.876,E2 -24528.876} C_VEL
LIN {X 0,Y 157.762,Z 688.991,A -85,B 0,C 180,E1 -24532.227,E2 -24532.227} C_VEL
LIN {X 0,Y 156.716,Z 691.066,A -85,B 0,C 180,E1 -24533.019,E2 -24533.019} C_VEL
LIN {X 0,Y 154.174,Z 694.798,A -85,B 0,C 180,E1 -24534.432,E2 -24534.432} C_VEL
LIN {X 0,Y 148.545,Z 700.401,A -85,B 0,C 180,E1 -24536.688,E2 -24536.688} C_VEL
LIN {X 0,Y 143.124,Z 705.599,A -85,B 0,C 180,E1 -24539.245,E2 -24539.245} C_VEL
LIN {X 0,Y 140.973,Z 708.574,A -85,B 0,C 180,E1 -24541.098,E2 -24541.098} C_VEL
LIN {X 0,Y 137.674,Z 716.007,A -85,B 0,C 180,E1 -24546.759,E2 -24546.759} C_VEL
LIN {X 0,Y 135.824,Z 721.294,A -85,B 0,C 180,E1 -24551.912,E2 -24551.912} C_VEL
LIN {X 0,Y 135.104,Z 726.112,A -85,B 0,C 180,E1 -24557.99,E2 -24557.99} C_VEL
LIN {X 0,Y 135.579,Z 729.589,A -85,B 0,C 180,E1 -24564.048,E2 -24564.048} C_VEL
LIN {X 0,Y 136.753,Z 731.692,A -85,B 0,C 180,E1 -24569.999,E2 -24569.999} C_VEL
LIN {X 0,Y 135.483,Z 732.042,A -85,B 0,C 180,E1 -24575.954,E2 -24575.954} C_VEL
LIN {X 0,Y 134.885,Z 731.18,A -85,B 0,C 180,E1 -24582.028,E2 -24582.028} C_VEL
LIN {X 0,Y 135.675,Z 729.208,A -85,B 0,C 180,E1 -24588.106,E2 -24588.106} C_VEL
LIN {X 0,Y 138.034,Z 726.112,A -85,B 0,C 180,E1 -24594.035,E2 -24594.035} C_VEL
LIN {X 0,Y 141.799,Z 721.789,A -85,B 0,C 180,E1 -24599.709,E2 -24599.709} C_VEL
LIN {X 0,Y 147.009,Z 716.223,A -85,B 0,C 180,E1 -24605.005,E2 -24605.005} C_VEL
LIN {X 0,Y 153.485,Z 709.277,A -85,B 0,C 180,E1 -24609.868,E2 -24609.868} C_VEL
LIN {X 0,Y 160.116,Z 701.939,A -85,B 0,C 180,E1 -24613.732,E2 -24613.732} C_VEL
LIN {X 0,Y 167.602,Z 693.251,A -85,B 0,C 180,E1 -24617.205,E2 -24617.205} C_VEL
LIN {X 0,Y 174.496,Z 684.502,A -85,B 0,C 180,E1 -24619.926,E2 -24619.926} C_VEL
LIN {X 0,Y 181.85,Z 674.245,A -85,B 0,C 180,E1 -24622.394,E2 -24622.394} C_VEL
LIN {X 0,Y 189.675,Z 662.154,A -85,B 0,C 180,E1 -24624.6,E2 -24624.6} C_VEL
LIN {X 0,Y 196.518,Z 650.147,A -85,B 0,C 180,E1 -24626.248,E2 -24626.248} C_VEL
LIN {X 0,Y 202.826,Z 637.207,A -85,B 0,C 180,E1 -24627.626,E2 -24627.626} C_VEL
LIN {X 0,Y 207.793,Z 625.097,A -85,B 0,C 180,E1 -24628.647,E2 -24628.647} C_VEL
LIN {X 0,Y 212.43,Z 611.196,A -85,B 0,C 180,E1 -24629.566,E2 -24629.566} C_VEL
LIN {X 0,Y 216.415,Z 595.567,A -85,B 0,C 180,E1 -24630.303,E2 -24630.303} C_VEL
LIN {X 0,Y 219.019,Z 580.16,A -85,B 0,C 180,E1 -24630.852,E2 -24630.852} C_VEL
LIN {X 0,Y 223.11,Z 536.684,A -85,B 0,C 180,E1 -24631.953,E2 -24631.953} C_VEL
LIN {X 0,Y 223.069,Z 528.989,A -85,B 0,C 180,E1 -24632.563,E2 -24632.563} C_VEL
LIN {X 0,Y 220.107,Z 519.51,A -85,B 0,C 180,E1 -24635.15,E2 -24635.15} C_VEL
LIN {X 0,Y 217.242,Z 511.083,A -85,B 0,C 180,E1 -24637.984,E2 -24637.984} C_VEL
LIN {X 0,Y 215.407,Z 506.03,A -85,B 0,C 180,E1 -24640.048,E2 -24640.048} C_VEL
LIN {X 0,Y 213.399,Z 500.572,A -85,B 0,C 180,E1 -24642.679,E2 -24642.679} C_VEL
LIN {X 0,Y 211.62,Z 495.553,A -85,B 0,C 180,E1 -24645.611,E2 -24645.611} C_VEL
LIN {X 0,Y 209.604,Z 489.439,A -85,B 0,C 180,E1 -24650.714,E2 -24650.714} C_VEL
LIN {X 0,Y 209.177,Z 487.665,A -85,B 0,C 180,E1 -24652.826,E2 -24652.826} C_VEL
LIN {X 0,Y 209.167,Z 487.501,A -85,B 0,C 180,E1 -24660,E2 -24660} C_VEL
LIN {X 0,Y 209.384,Z 488.248,A -85,B 0,C 180,E1 -24661.172,E2 -24661.172} C_VEL
LIN {X 0,Y 211.615,Z 492.387,A -85,B 0,C 180,E1 -24666.795,E2 -24666.795} C_VEL
LIN {X 0,Y 214.137,Z 496.973,A -85,B 0,C 180,E1 -24670.617,E2 -24670.617} C_VEL
LIN {X 0,Y 216.23,Z 500.69,A -85,B 0,C 180,E1 -24673.069,E2 -24673.069} C_VEL
LIN {X 0,Y 219.579,Z 506.612,A -85,B 0,C 180,E1 -24676.313,E2 -24676.313} C_VEL
LIN {X 0,Y 223.735,Z 514.73,A -85,B 0,C 180,E1 -24679.699,E2 -24679.699} C_VEL
LIN {X 0,Y 224.783,Z 516.918,A -85,B 0,C 180,E1 -24680.475,E2 -24680.475} C_VEL
LIN {X 0,Y 221.795,Z 552.618,A -85,B 0,C 180,E1 -24681.611,E2 -24681.611} C_VEL
LIN {X 0,Y 219.497,Z 568.257,A -85,B 0,C 180,E1 -24682.409,E2 -24682.409} C_VEL
LIN {X 0,Y 216.26,Z 582.519,A -85,B 0,C 180,E1 -24683.352,E2 -24683.352} C_VEL
LIN {X 0,Y 212.397,Z 595.578,A -85,B 0,C 180,E1 -24684.507,E2 -24684.507} C_VEL
LIN {X 0,Y 207.764,Z 608.304,A -85,B 0,C 180,E1 -24685.938,E2 -24685.938} C_VEL
LIN {X 0,Y 202.235,Z 620.658,A -85,B 0,C 180,E1 -24687.609,E2 -24687.609} C_VEL
LIN {X 0,Y 196.041,Z 632.427,A -85,B 0,C 180,E1 -24689.62,E2 -24689.62} C_VEL
LIN {X 0,Y 188.857,Z 644.122,A -85,B 0,C 180,E1 -24692.16,E2 -24692.16} C_VEL
LIN {X 0,Y 181.997,Z 653.864,A -85,B 0,C 180,E1 -24694.86,E2 -24694.86} C_VEL
LIN {X 0,Y 174.396,Z 663.307,A -85,B 0,C 180,E1 -24698.206,E2 -24698.206} C_VEL
LIN {X 0,Y 168.344,Z 670.095,A -85,B 0,C 180,E1 -24701.286,E2 -24701.286} C_VEL
LIN {X 0,Y 162.679,Z 675.754,A -85,B 0,C 180,E1 -24704.537,E2 -24704.537} C_VEL
LIN {X 0,Y 155.929,Z 681.916,A -85,B 0,C 180,E1 -24709.194,E2 -24709.194} C_VEL
LIN {X 0,Y 150.104,Z 686.614,A -85,B 0,C 180,E1 -24714.181,E2 -24714.181} C_VEL
LIN {X 0,Y 146.426,Z 689.291,A -85,B 0,C 180,E1 -24718.134,E2 -24718.134} C_VEL
LIN {X 0,Y 142.456,Z 691.72,A -85,B 0,C 180,E1 -24723.642,E2 -24723.642} C_VEL
LIN {X 0,Y 139.585,Z 692.985,A -85,B 0,C 180,E1 -24729.365,E2 -24729.365} C_VEL
LIN {X 0,Y 137.843,Z 693.083,A -85,B 0,C 180,E1 -24735.637,E2 -24735.637} C_VEL
LIN {X 0,Y 137.144,Z 692.178,A -85,B 0,C 180,E1 -24741.158,E2 -24741.158} C_VEL
LIN {X 0,Y 137.481,Z 690.128,A -85,B 0,C 180,E1 -24747.071,E2 -24747.071} C_VEL
LIN {X 0,Y 138.828,Z 686.895,A -85,B 0,C 180,E1 -24752.903,E2 -24752.903} C_VEL
LIN {X 0,Y 141.115,Z 682.467,A -85,B 0,C 180,E1 -24758.594,E2 -24758.594} C_VEL
LIN {X 0,Y 144.416,Z 676.734,A -85,B 0,C 180,E1 -24764.084,E2 -24764.084} C_VEL
LIN {X 0,Y 148.685,Z 669.532,A -85,B 0,C 180,E1 -24769.322,E2 -24769.322} C_VEL
LIN {X 0,Y 153.147,Z 661.836,A -85,B 0,C 180,E1 -24773.675,E2 -24773.675} C_VEL
LIN {X 0,Y 158.285,Z 652.604,A -85,B 0,C 180,E1 -24777.789,E2 -24777.789} C_VEL
LIN {X 0,Y 163.173,Z 643.211,A -85,B 0,C 180,E1 -24781.121,E2 -24781.121} C_VEL
LIN {X 0,Y 168.336,Z 632.097,A -85,B 0,C 180,E1 -24784.307,E2 -24784.307} C_VEL
LIN {X 0,Y 173.281,Z 619.914,A -85,B 0,C 180,E1 -24787.107,E2 -24787.107} C_VEL
LIN {X 0,Y 177.704,Z 607.907,A -85,B 0,C 180,E1 -24789.256,E2 -24789.256} C_VEL
LIN {X 0,Y 181.66,Z 594.934,A -85,B 0,C 180,E1 -24791.124,E2 -24791.124} C_VEL
LIN {X 0,Y 185.174,Z 580.687,A -85,B 0,C 180,E1 -24792.72,E2 -24792.72} C_VEL
LIN {X 0,Y 188.117,Z 565.147,A -85,B 0,C 180,E1 -24794,E2 -24794} C_VEL
LIN {X 0,Y 190.029,Z 549.747,A -85,B 0,C 180,E1 -24794.895,E2 -24794.895} C_VEL
LIN {X 0,Y 192.446,Z 513.19,A -85,B 0,C 180,E1 -24796.243,E2 -24796.243} C_VEL
LIN {X 0,Y 193.907,Z 492.628,A -85,B 0,C 180,E1 -24796.914,E2 -24796.914} C_VEL
LIN {X 0,Y 189.124,Z 482.873,A -85,B 0,C 180,E1 -24799.507,E2 -24799.507} C_VEL
LIN {X 0,Y 184.556,Z 474.515,A -85,B 0,C 180,E1 -24802.22,E2 -24802.22} C_VEL
LIN {X 0,Y 179.836,Z 466.637,A -85,B 0,C 180,E1 -24805.355,E2 -24805.355} C_VEL
LIN {X 0,Y 175.884,Z 460.642,A -85,B 0,C 180,E1 -24808.334,E2 -24808.334} C_VEL
LIN {X 0,Y 173.683,Z 457.326,A -85,B 0,C 180,E1 -24810.205,E2 -24810.205} C_VEL
LIN {X 0,Y 170.843,Z 453.286,A -85,B 0,C 180,E1 -24812.897,E2 -24812.897} C_VEL
LIN {X 0,Y 168.203,Z 449.426,A -85,B 0,C 180,E1 -24815.835,E2 -24815.835} C_VEL
LIN {X 0,Y 165.156,Z 445.742,A -85,B 0,C 180,E1 -24819.936,E2 -24819.936} C_VEL
LIN {X 0,Y 164.28,Z 444.099,A -85,B 0,C 180,E1 -24821.491,E2 -24821.491} C_VEL
LIN {X 0,Y 161.74,Z 441.668,A -85,B 0,C 180,E1 -24827.132,E2 -24827.132} C_VEL
LIN {X 0,Y 160.975,Z 438.741,A -85,B 0,C 180,E1 -24831.701,E2 -24831.701} C_VEL
LIN {X 0,Y 161.243,Z 438.859,A -85,B 0,C 180,E1 -24838.875,E2 -24838.875} C_VEL
LIN {X 0,Y 162.071,Z 441.801,A -85,B 0,C 180,E1 -24842.718,E2 -24842.718} C_VEL
LIN {X 0,Y 164.673,Z 444.339,A -85,B 0,C 180,E1 -24848.049,E2 -24848.049} C_VEL
LIN {X 0,Y 166.743,Z 447.867,A -85,B 0,C 180,E1 -24851.292,E2 -24851.292} C_VEL
LIN {X 0,Y 168.389,Z 449.657,A -85,B 0,C 180,E1 -24853.308,E2 -24853.308} C_VEL
LIN {X 0,Y 171.863,Z 455.81,A -85,B 0,C 180,E1 -24857.15,E2 -24857.15} C_VEL
LIN {X 0,Y 175.41,Z 462.87,A -85,B 0,C 180,E1 -24860.465,E2 -24860.465} C_VEL
LIN {X 0,Y 178.703,Z 469.838,A -85,B 0,C 180,E1 -24863.158,E2 -24863.158} C_VEL
LIN {X 0,Y 183.173,Z 480.214,A -85,B 0,C 180,E1 -24866.416,E2 -24866.416} C_VEL
LIN {X 0,Y 187.557,Z 491.808,A -85,B 0,C 180,E1 -24869.305,E2 -24869.305} C_VEL
LIN {X 0,Y 190.775,Z 501.336,A -85,B 0,C 180,E1 -24871.285,E2 -24871.285} C_VEL
LIN {X 0,Y 191.582,Z 530.711,A -85,B 0,C 180,E1 -24873.384,E2 -24873.384} C_VEL
LIN {X 0,Y 187.34,Z 584.61,A -85,B 0,C 180,E1 -24875.087,E2 -24875.087} C_VEL
LIN {X 0,Y 184.898,Z 600.704,A -85,B 0,C 180,E1 -24875.896,E2 -24875.896} C_VEL
LIN {X 0,Y 181.542,Z 616.026,A -85,B 0,C 180,E1 -24877.018,E2 -24877.018} C_VEL
LIN {X 0,Y 177.244,Z 630.734,A -85,B 0,C 180,E1 -24878.453,E2 -24878.453} C_VEL
LIN {X 0,Y 172.507,Z 644.159,A -85,B 0,C 180,E1 -24880.193,E2 -24880.193} C_VEL
LIN {X 0,Y 166.947,Z 657.389,A -85,B 0,C 180,E1 -24882.397,E2 -24882.397} C_VEL
LIN {X 0,Y 162.95,Z 665.933,A -85,B 0,C 180,E1 -24884.19,E2 -24884.19} C_VEL
LIN {X 0,Y 157.568,Z 677.164,A -85,B 0,C 180,E1 -24887.141,E2 -24887.141} C_VEL
LIN {X 0,Y 152.108,Z 687.52,A -85,B 0,C 180,E1 -24890.557,E2 -24890.557} C_VEL
LIN {X 0,Y 146.638,Z 697.688,A -85,B 0,C 180,E1 -24894.891,E2 -24894.891} C_VEL
LIN {X 0,Y 142.186,Z 706.217,A -85,B 0,C 180,E1 -24899.559,E2 -24899.559} C_VEL
LIN {X 0,Y 140.973,Z 708.574,A -85,B 0,C 180,E1 -24901.098,E2 -24901.098} C_VEL
LIN {X 0,Y 138.957,Z 711.433,A -85,B 0,C 180,E1 -24903.051,E2 -24903.051} C_VEL
LIN {X 0,Y 134.251,Z 715.529,A -85,B 0,C 180,E1 -24906.289,E2 -24906.289} C_VEL
LIN {X 0,Y 129.957,Z 719.161,A -85,B 0,C 180,E1 -24909.852,E2 -24909.852} C_VEL
LIN {X 0,Y 128.648,Z 721.189,A -85,B 0,C 180,E1 -24912.24,E2 -24912.24} C_VEL
LIN {X 0,Y 128.064,Z 724.944,A -85,B 0,C 180,E1 -24917.319,E2 -24917.319} C_VEL
LIN {X 0,Y 128.485,Z 728.474,A -85,B 0,C 180,E1 -24923.718,E2 -24923.718} C_VEL
LIN {X 0,Y 129.679,Z 730.615,A -85,B 0,C 180,E1 -24929.999,E2 -24929.999} C_VEL
LIN {X 0,Y 128.372,Z 730.997,A -85,B 0,C 180,E1 -24936.285,E2 -24936.285} C_VEL
LIN {X 0,Y 127.849,Z 730.173,A -85,B 0,C 180,E1 -24942.701,E2 -24942.701} C_VEL
LIN {X 0,Y 128.854,Z 728.248,A -85,B 0,C 180,E1 -24949.1,E2 -24949.1} C_VEL
LIN {X 0,Y 131.484,Z 725.173,A -85,B 0,C 180,E1 -24955.314,E2 -24955.314} C_VEL
LIN {X 0,Y 135.567,Z 720.895,A -85,B 0,C 180,E1 -24961.224,E2 -24961.224} C_VEL
LIN {X 0,Y 141.157,Z 715.383,A -85,B 0,C 180,E1 -24966.686,E2 -24966.686} C_VEL
LIN {X 0,Y 148.02,Z 708.496,A -85,B 0,C 180,E1 -24971.658,E2 -24971.658} C_VEL
LIN {X 0,Y 156.109,Z 700.072,A -85,B 0,C 180,E1 -24976.078,E2 -24976.078} C_VEL
LIN {X 0,Y 164.045,Z 691.225,A -85,B 0,C 180,E1 -24979.5,E2 -24979.5} C_VEL
LIN {X 0,Y 171.249,Z 682.333,A -85,B 0,C 180,E1 -24982.183,E2 -24982.183} C_VEL
LIN {X 0,Y 178.918,Z 671.919,A -85,B 0,C 180,E1 -24984.591,E2 -24984.591} C_VEL
LIN {X 0,Y 187.04,Z 659.582,A -85,B 0,C 180,E1 -24986.721,E2 -24986.721} C_VEL
LIN {X 0,Y 194.795,Z 645.931,A -85,B 0,C 180,E1 -24988.466,E2 -24988.466} C_VEL
LIN {X 0,Y 201.23,Z 632.307,A -85,B 0,C 180,E1 -24989.81,E2 -24989.81} C_VEL
LIN {X 0,Y 206.763,Z 618.262,A -85,B 0,C 180,E1 -24990.82,E2 -24990.82} C_VEL
LIN {X 0,Y 211.52,Z 602.534,A -85,B 0,C 180,E1 -24991.698,E2 -24991.698} C_VEL
LIN {X 0,Y 214.909,Z 586.856,A -85,B 0,C 180,E1 -24992.33,E2 -24992.33} C_VEL
LIN {X 0,Y 217.052,Z 570.348,A -85,B 0,C 180,E1 -24992.814,E2 -24992.814} C_VEL
LIN {X 0,Y 220.115,Z 537.786,A -85,B 0,C 180,E1 -24993.604,E2 -24993.604} C_VEL
LIN {X 0,Y 220.121,Z 532.654,A -85,B 0,C 180,E1 -24994.023,E2 -24994.023} C_VEL
LIN {X 0,Y 217.39,Z 523.464,A -85,B 0,C 180,E1 -24996.662,E2 -24996.662} C_VEL
LIN {X 0,Y 214.953,Z 515.857,A -85,B 0,C 180,E1 -24999.341,E2 -24999.341} C_VEL
LIN {X 0,Y 213.378,Z 511.276,A -85,B 0,C 180,E1 -25001.308,E2 -25001.308} C_VEL
LIN {X 0,Y 211.817,Z 506.632,A -85,B 0,C 180,E1 -25003.591,E2 -25003.591} C_VEL
LIN {X 0,Y 210.299,Z 502.004,A -85,B 0,C 180,E1 -25006.348,E2 -25006.348} C_VEL
LIN {X 0,Y 208.575,Z 496.211,A -85,B 0,C 180,E1 -25011.249,E2 -25011.249} C_VEL
LIN {X 0,Y 208.194,Z 494.698,A -85,B 0,C 180,E1 -25013.342,E2 -25013.342} C_VEL
LIN {X 0,Y 208.294,Z 494.557,A -85,B 0,C 180,E1 -25020,E2 -25020} C_VEL
LIN {X 0,Y 210.481,Z 499.289,A -85,B 0,C 180,E1 -25026.387,E2 -25026.387} C_VEL
LIN {X 0,Y 212.724,Z 503.528,A -85,B 0,C 180,E1 -25029.989,E2 -25029.989} C_VEL
LIN {X 0,Y 214.864,Z 507.534,A -85,B 0,C 180,E1 -25032.636,E2 -25032.636} C_VEL
LIN {X 0,Y 217.915,Z 513.218,A -85,B 0,C 180,E1 -25035.731,E2 -25035.731} C_VEL
LIN {X 0,Y 221.617,Z 520.784,A -85,B 0,C 180,E1 -25038.909,E2 -25038.909} C_VEL
LIN {X 0,Y 218.662,Z 554.504,A -85,B 0,C 180,E1 -25040.004,E2 -25040.004} C_VEL
LIN {X 0,Y 216.35,Z 569.44,A -85,B 0,C 180,E1 -25040.766,E2 -25040.766} C_VEL
LIN {X 0,Y 212.721,Z 584.735,A -85,B 0,C 180,E1 -25041.787,E2 -25041.787} C_VEL
LIN {X 0,Y 208.844,Z 597.279,A -85,B 0,C 180,E1 -25042.9,E2 -25042.9} C_VEL
LIN {X 0,Y 203.395,Z 611.437,A -85,B 0,C 180,E1 -25044.497,E2 -25044.497} C_VEL
LIN {X 0,Y 197.703,Z 623.399,A -85,B 0,C 180,E1 -25046.161,E2 -25046.161} C_VEL
LIN {X 0,Y 191.304,Z 634.862,A -85,B 0,C 180,E1 -25048.157,E2 -25048.157} C_VEL
LIN {X 0,Y 183.907,Z 646.313,A -85,B 0,C 180,E1 -25050.706,E2 -25050.706} C_VEL
LIN {X 0,Y 176.818,Z 655.856,A -85,B 0,C 180,E1 -25053.421,E2 -25053.421} C_VEL
LIN {X 0,Y 168.94,Z 665.13,A -85,B 0,C 180,E1 -25056.796,E2 -25056.796} C_VEL
LIN {X 0,Y 161.645,Z 672.744,A -85,B 0,C 180,E1 -25060.45,E2 -25060.45} C_VEL
LIN {X 0,Y 154.019,Z 679.791,A -85,B 0,C 180,E1 -25064.989,E2 -25064.989} C_VEL
LIN {X 0,Y 147.794,Z 684.914,A -85,B 0,C 180,E1 -25069.54,E2 -25069.54} C_VEL
LIN {X 0,Y 142.951,Z 688.471,A -85,B 0,C 180,E1 -25073.848,E2 -25073.848} C_VEL
LIN {X 0,Y 138.093,Z 691.564,A -85,B 0,C 180,E1 -25079.409,E2 -25079.409} C_VEL
LIN {X 0,Y 134.309,Z 693.464,A -85,B 0,C 180,E1 -25085.255,E2 -25085.255} C_VEL
LIN {X 0,Y 131.802,Z 694.209,A -85,B 0,C 180,E1 -25091.343,E2 -25091.343} C_VEL
LIN {X 0,Y 130.497,Z 693.841,A -85,B 0,C 180,E1 -25097.561,E2 -25097.561} C_VEL
LIN {X 0,Y 130.12,Z 692.411,A -85,B 0,C 180,E1 -25103.8,E2 -25103.8} C_VEL
LIN {X 0,Y 130.96,Z 689.803,A -85,B 0,C 180,E1 -25110.001,E2 -25110.001} C_VEL
LIN {X 0,Y 132.886,Z 686.024,A -85,B 0,C 180,E1 -25116.073,E2 -25116.073} C_VEL
LIN {X 0,Y 135.769,Z 681.024,A -85,B 0,C 180,E1 -25121.951,E2 -25121.951} C_VEL
LIN {X 0,Y 139.757,Z 674.64,A -85,B 0,C 180,E1 -25127.562,E2 -25127.562} C_VEL
LIN {X 0,Y 144.693,Z 666.695,A -85,B 0,C 180,E1 -25132.866,E2 -25132.866} C_VEL
LIN {X 0,Y 149.768,Z 658.231,A -85,B 0,C 180,E1 -25137.228,E2 -25137.228} C_VEL
LIN {X 0,Y 155.503,Z 648.06,A -85,B 0,C 180,E1 -25141.315,E2 -25141.315} C_VEL
LIN {X 0,Y 160.826,Z 637.652,A -85,B 0,C 180,E1 -25144.617,E2 -25144.617} C_VEL
LIN {X 0,Y 166.313,Z 625.246,A -85,B 0,C 180,E1 -25147.788,E2 -25147.788} C_VEL
LIN {X 0,Y 171.358,Z 612.664,A -85,B 0,C 180,E1 -25150.238,E2 -25150.238} C_VEL
LIN {X 0,Y 175.994,Z 598.822,A -85,B 0,C 180,E1 -25152.366,E2 -25152.366} C_VEL
LIN {X 0,Y 179.907,Z 584.283,A -85,B 0,C 180,E1 -25154.094,E2 -25154.094} C_VEL
LIN {X 0,Y 182.921,Z 569.69,A -85,B 0,C 180,E1 -25155.397,E2 -25155.397} C_VEL
LIN {X 0,Y 185.189,Z 554.468,A -85,B 0,C 180,E1 -25156.344,E2 -25156.344} C_VEL
LIN {X 0,Y 186.619,Z 535.588,A -85,B 0,C 180,E1 -25157.174,E2 -25157.174} C_VEL
LIN {X 0,Y 189.509,Z 495.595,A -85,B 0,C 180,E1 -25158.515,E2 -25158.515} C_VEL
LIN {X 0,Y 184.567,Z 485.345,A -85,B 0,C 180,E1 -25161.439,E2 -25161.439} C_VEL
LIN {X 0,Y 178.644,Z 474.641,A -85,B 0,C 180,E1 -25165.392,E2 -25165.392} C_VEL
LIN {X 0,Y 173.953,Z 467.16,A -85,B 0,C 180,E1 -25169.048,E2 -25169.048} C_VEL
LIN {X 0,Y 171.497,Z 463.402,A -85,B 0,C 180,E1 -25171.25,E2 -25171.25} C_VEL
LIN {X 0,Y 168.996,Z 459.63,A -85,B 0,C 180,E1 -25173.788,E2 -25173.788} C_VEL
LIN {X 0,Y 166.324,Z 455.666,A -85,B 0,C 180,E1 -25176.97,E2 -25176.97} C_VEL
LIN {X 0,Y 163.859,Z 452.528,A -85,B 0,C 180,E1 -25180.537,E2 -25180.537} C_VEL
LIN {X 0,Y 163.139,Z 451.027,A -85,B 0,C 180,E1 -25181.903,E2 -25181.903} C_VEL
LIN {X 0,Y 160.697,Z 448.515,A -85,B 0,C 180,E1 -25187.689,E2 -25187.689} C_VEL
LIN {X 0,Y 160.067,Z 445.755,A -85,B 0,C 180,E1 -25192.042,E2 -25192.042} C_VEL
LIN {X 0,Y 160.286,Z 445.773,A -85,B 0,C 180,E1 -25198.366,E2 -25198.366} C_VEL
LIN {X 0,Y 161.007,Z 448.677,A -85,B 0,C 180,E1 -25202.188,E2 -25202.188} C_VEL
LIN {X 0,Y 163.385,Z 451.128,A -85,B 0,C 180,E1 -25207.414,E2 -25207.414} C_VEL
LIN {X 0,Y 165.492,Z 454.74,A -85,B 0,C 180,E1 -25210.862,E2 -25210.862} C_VEL
LIN {X 0,Y 166.855,Z 456.335,A -85,B 0,C 180,E1 -25212.62,E2 -25212.62} C_VEL
LIN {X 0,Y 169.804,Z 461.88,A -85,B 0,C 180,E1 -25216.108,E2 -25216.108} C_VEL
LIN {X 0,Y 173.091,Z 468.841,A -85,B 0,C 180,E1 -25219.416,E2 -25219.416} C_VEL
LIN {X 0,Y 176.079,Z 475.447,A -85,B 0,C 180,E1 -25222.032,E2 -25222.032} C_VEL
LIN {X 0,Y 180.36,Z 485.976,A -85,B 0,C 180,E1 -25225.38,E2 -25225.38} C_VEL
LIN {X 0,Y 184.778,Z 498.349,A -85,B 0,C 180,E1 -25228.484,E2 -25228.484} C_VEL
LIN {X 0,Y 186.63,Z 504.328,A -85,B 0,C 180,E1 -25229.725,E2 -25229.725} C_VEL
LIN {X 0,Y 187.128,Z 532.615,A -85,B 0,C 180,E1 -25231.757,E2 -25231.757} C_VEL
LIN {X 0,Y 182.966,Z 583.177,A -85,B 0,C 180,E1 -25233.338,E2 -25233.338} C_VEL
LIN {X 0,Y 180.635,Z 598.656,A -85,B 0,C 180,E1 -25234.107,E2 -25234.107} C_VEL
LIN {X 0,Y 177.288,Z 613.639,A -85,B 0,C 180,E1 -25235.155,E2 -25235.155} C_VEL
LIN {X 0,Y 172.854,Z 628.666,A -85,B 0,C 180,E1 -25236.582,E2 -25236.582} C_VEL
LIN {X 0,Y 168.592,Z 640.673,A -85,B 0,C 180,E1 -25238.11,E2 -25238.11} C_VEL
LIN {X 0,Y 163.202,Z 653.353,A -85,B 0,C 180,E1 -25240.108,E2 -25240.108} C_VEL
LIN {X 0,Y 157.981,Z 664.268,A -85,B 0,C 180,E1 -25242.304,E2 -25242.304} C_VEL
LIN {X 0,Y 152.347,Z 675.608,A -85,B 0,C 180,E1 -25245.291,E2 -25245.291} C_VEL
LIN {X 0,Y 146.615,Z 686.056,A -85,B 0,C 180,E1 -25248.768,E2 -25248.768} C_VEL
LIN {X 0,Y 140.788,Z 696.293,A -85,B 0,C 180,E1 -25253.199,E2 -25253.199} C_VEL
LIN {X 0,Y 135.973,Z 704.867,A -85,B 0,C 180,E1 -25258.008,E2 -25258.008} C_VEL
LIN {X 0,Y 132.299,Z 711.998,A -85,B 0,C 180,E1 -25263.157,E2 -25263.157} C_VEL
LIN {X 0,Y 129.459,Z 718.647,A -85,B 0,C 180,E1 -25269.336,E2 -25269.336} C_VEL
LIN {X 0,Y 128.648,Z 721.189,A -85,B 0,C 180,E1 -25272.24,E2 -25272.24} C_VEL
LIN {X 0,Y 127.561,Z 723.073,A -85,B 0,C 180,E1 -25274.699,E2 -25274.699} C_VEL
LIN {X 0,Y 124.497,Z 725.484,A -85,B 0,C 180,E1 -25278.848,E2 -25278.848} C_VEL
LIN {X 0,Y 122.299,Z 727.008,A -85,B 0,C 180,E1 -25282.35,E2 -25282.35} C_VEL
LIN {X 0,Y 121.628,Z 728.018,A -85,B 0,C 180,E1 -25285.09,E2 -25285.09} C_VEL
LIN {X 0,Y 121.7,Z 728.339,A -85,B 0,C 180,E1 -25286.011,E2 -25286.011} C_VEL
LIN {X 0,Y 122.603,Z 729.537,A -85,B 0,C 180,E1 -25289.999,E2 -25289.999} C_VEL
LIN {X 0,Y 121.273,Z 729.954,A -85,B 0,C 180,E1 -25296.654,E2 -25296.654} C_VEL
LIN {X 0,Y 120.858,Z 729.17,A -85,B 0,C 180,E1 -25303.449,E2 -25303.449} C_VEL
LIN {X 0,Y 122.083,Z 727.287,A -85,B 0,C 180,E1 -25310.205,E2 -25310.205} C_VEL
LIN {X 0,Y 124.997,Z 724.233,A -85,B 0,C 180,E1 -25316.729,E2 -25316.729} C_VEL
LIN {X 0,Y 129.444,Z 720.005,A -85,B 0,C 180,E1 -25322.882,E2 -25322.882} C_VEL
LIN {X 0,Y 135.452,Z 714.549,A -85,B 0,C 180,E1 -25328.505,E2 -25328.505} C_VEL
LIN {X 0,Y 142.732,Z 707.719,A -85,B 0,C 180,E1 -25333.576,E2 -25333.576} C_VEL
LIN {X 0,Y 150.088,Z 700.513,A -85,B 0,C 180,E1 -25337.516,E2 -25337.516} C_VEL
LIN {X 0,Y 158.262,Z 691.968,A -85,B 0,C 180,E1 -25340.995,E2 -25340.995} C_VEL
LIN {X 0,Y 166.964,Z 681.765,A -85,B 0,C 180,E1 -25344.12,E2 -25344.12} C_VEL
LIN {X 0,Y 174.88,Z 671.402,A -85,B 0,C 180,E1 -25346.497,E2 -25346.497} C_VEL
LIN {X 0,Y 183.233,Z 659.178,A -85,B 0,C 180,E1 -25348.581,E2 -25348.581} C_VEL
LIN {X 0,Y 190.458,Z 646.997,A -85,B 0,C 180,E1 -25350.126,E2 -25350.126} C_VEL
LIN {X 0,Y 197.033,Z 633.827,A -85,B 0,C 180,E1 -25351.44,E2 -25351.44} C_VEL
LIN {X 0,Y 203.032,Z 619.416,A -85,B 0,C 180,E1 -25352.496,E2 -25352.496} C_VEL
LIN {X 0,Y 207.529,Z 605.725,A -85,B 0,C 180,E1 -25353.272,E2 -25353.272} C_VEL
LIN {X 0,Y 211.23,Z 590.586,A -85,B 0,C 180,E1 -25353.936,E2 -25353.936} C_VEL
LIN {X 0,Y 213.726,Z 575.152,A -85,B 0,C 180,E1 -25354.422,E2 -25354.422} C_VEL
LIN {X 0,Y 217.351,Z 538.449,A -85,B 0,C 180,E1 -25355.315,E2 -25355.315} C_VEL
LIN {X 0,Y 217.303,Z 536.314,A -85,B 0,C 180,E1 -25355.539,E2 -25355.539} C_VEL
LIN {X 0,Y 214.748,Z 527.106,A -85,B 0,C 180,E1 -25358.309,E2 -25358.309} C_VEL
LIN {X 0,Y 212.469,Z 519.507,A -85,B 0,C 180,E1 -25361.169,E2 -25361.169} C_VEL
LIN {X 0,Y 210.343,Z 512.908,A -85,B 0,C 180,E1 -25364.414,E2 -25364.414} C_VEL
LIN {X 0,Y 209.083,Z 508.643,A -85,B 0,C 180,E1 -25366.949,E2 -25366.949} C_VEL
LIN {X 0,Y 207.583,Z 503.026,A -85,B 0,C 180,E1 -25371.712,E2 -25371.712} C_VEL
LIN {X 0,Y 207.289,Z 501.732,A -85,B 0,C 180,E1 -25373.531,E2 -25373.531} C_VEL
LIN {X 0,Y 207.245,Z 501.516,A -85,B 0,C 180,E1 -25379.029,E2 -25379.029} C_VEL
LIN {X 0,Y 207.453,Z 501.931,A -85,B 0,C 180,E1 -25380.304,E2 -25380.304} C_VEL
LIN {X 0,Y 209.326,Z 506.084,A -85,B 0,C 180,E1 -25385.902,E2 -25385.902} C_VEL
LIN {X 0,Y 211.428,Z 510.312,A -85,B 0,C 180,E1 -25389.491,E2 -25389.491} C_VEL
LIN {X 0,Y 213.541,Z 514.436,A -85,B 0,C 180,E1 -25392.232,E2 -25392.232} C_VEL
LIN {X 0,Y 216.788,Z 520.856,A -85,B 0,C 180,E1 -25395.634,E2 -25395.634} C_VEL
LIN {X 0,Y 218.589,Z 524.725,A -85,B 0,C 180,E1 -25397.284,E2 -25397.284} C_VEL
LIN {X 0,Y 215.806,Z 555.56,A -85,B 0,C 180,E1 -25398.311,E2 -25398.311} C_VEL
LIN {X 0,Y 213.466,Z 570.264,A -85,B 0,C 180,E1 -25399.058,E2 -25399.058} C_VEL
LIN {X 0,Y 210.028,Z 584.537,A -85,B 0,C 180,E1 -25399.978,E2 -25399.978} C_VEL
LIN {X 0,Y 205.784,Z 597.973,A -85,B 0,C 180,E1 -25401.133,E2 -25401.133} C_VEL
LIN {X 0,Y 200.818,Z 610.688,A -85,B 0,C 180,E1 -25402.537,E2 -25402.537} C_VEL
LIN {X 0,Y 195.296,Z 622.275,A -85,B 0,C 180,E1 -25404.06,E2 -25404.06} C_VEL
LIN {X 0,Y 188.67,Z 634.117,A -85,B 0,C 180,E1 -25406.022,E2 -25406.022} C_VEL
LIN {X 0,Y 181.601,Z 644.984,A -85,B 0,C 180,E1 -25408.311,E2 -25408.311} C_VEL
LIN {X 0,Y 174.153,Z 654.928,A -85,B 0,C 180,E1 -25410.961,E2 -25410.961} C_VEL
LIN {X 0,Y 165.877,Z 664.541,A -85,B 0,C 180,E1 -25414.294,E2 -25414.294} C_VEL
LIN {X 0,Y 158.027,Z 672.565,A -85,B 0,C 180,E1 -25417.977,E2 -25417.977} C_VEL
LIN {X 0,Y 150.936,Z 678.964,A -85,B 0,C 180,E1 -25421.844,E2 -25421.844} C_VEL
LIN {X 0,Y 143.582,Z 684.869,A -85,B 0,C 180,E1 -25426.746,E2 -25426.746} C_VEL
LIN {X 0,Y 137.208,Z 689.326,A -85,B 0,C 180,E1 -25432.076,E2 -25432.076} C_VEL
LIN {X 0,Y 131.951,Z 692.476,A -85,B 0,C 180,E1 -25437.819,E2 -25437.819} C_VEL
LIN {X 0,Y 127.835,Z 694.429,A -85,B 0,C 180,E1 -25443.91,E2 -25443.91} C_VEL
LIN {X 0,Y 125.045,Z 695.227,A -85,B 0,C 180,E1 -25450.294,E2 -25450.294} C_VEL
LIN {X 0,Y 123.566,Z 694.907,A -85,B 0,C 180,E1 -25456.851,E2 -25456.851} C_VEL
LIN {X 0,Y 123.07,Z 693.511,A -85,B 0,C 180,E1 -25463.443,E2 -25463.443} C_VEL
LIN {X 0,Y 123.912,Z 690.94,A -85,B 0,C 180,E1 -25470.001,E2 -25470.001} C_VEL
LIN {X 0,Y 125.894,Z 687.216,A -85,B 0,C 180,E1 -25476.411,E2 -25476.411} C_VEL
LIN {X 0,Y 128.908,Z 682.274,A -85,B 0,C 180,E1 -25482.597,E2 -25482.597} C_VEL
LIN {X 0,Y 133.101,Z 675.95,A -85,B 0,C 180,E1 -25488.471,E2 -25488.471} C_VEL
LIN {X 0,Y 138.29,Z 668.072,A -85,B 0,C 180,E1 -25493.99,E2 -25493.99} C_VEL
LIN {X 0,Y 143.582,Z 659.69,A -85,B 0,C 180,E1 -25498.506,E2 -25498.506} C_VEL
LIN {X 0,Y 149.602,Z 649.604,A -85,B 0,C 180,E1 -25502.701,E2 -25502.701} C_VEL
LIN {X 0,Y 155.142,Z 639.307,A -85,B 0,C 180,E1 -25506.079,E2 -25506.079} C_VEL
LIN {X 0,Y 160.899,Z 627.022,A -85,B 0,C 180,E1 -25509.298,E2 -25509.298} C_VEL
LIN {X 0,Y 166.125,Z 614.612,A -85,B 0,C 180,E1 -25511.783,E2 -25511.783} C_VEL
LIN {X 0,Y 170.941,Z 600.998,A -85,B 0,C 180,E1 -25513.931,E2 -25513.931} C_VEL
LIN {X 0,Y 174.751,Z 587.877,A -85,B 0,C 180,E1 -25515.549,E2 -25515.549} C_VEL
LIN {X 0,Y 177.991,Z 573.468,A -85,B 0,C 180,E1 -25516.926,E2 -25516.926} C_VEL
LIN {X 0,Y 180.442,Z 558.856,A -85,B 0,C 180,E1 -25517.916,E2 -25517.916} C_VEL
LIN {X 0,Y 181.974,Z 542.45,A -85,B 0,C 180,E1 -25518.705,E2 -25518.705} C_VEL
LIN {X 0,Y 184.998,Z 501.819,A -85,B 0,C 180,E1 -25520.091,E2 -25520.091} C_VEL
LIN {X 0,Y 185.152,Z 498.375,A -85,B 0,C 180,E1 -25520.255,E2 -25520.255} C_VEL
LIN {X 0,Y 180.467,Z 488.647,A -85,B 0,C 180,E1 -25523.271,E2 -25523.271} C_VEL
LIN {X 0,Y 175.742,Z 479.874,A -85,B 0,C 180,E1 -25526.703,E2 -25526.703} C_VEL
LIN {X 0,Y 171.769,Z 473.246,A -85,B 0,C 180,E1 -25530.028,E2 -25530.028} C_VEL
LIN {X 0,Y 169.232,Z 469.228,A -85,B 0,C 180,E1 -25532.468,E2 -25532.468} C_VEL
LIN {X 0,Y 167.136,Z 465.953,A -85,B 0,C 180,E1 -25534.754,E2 -25534.754} C_VEL
LIN {X 0,Y 164.843,Z 462.383,A -85,B 0,C 180,E1 -25537.667,E2 -25537.667} C_VEL
LIN {X 0,Y 162.305,Z 458.726,A -85,B 0,C 180,E1 -25541.683,E2 -25541.683} C_VEL
LIN {X 0,Y 162.006,Z 457.961,A -85,B 0,C 180,E1 -25542.321,E2 -25542.321} C_VEL
LIN {X 0,Y 159.6,Z 455.175,A -85,B 0,C 180,E1 -25548.57,E2 -25548.57} C_VEL
LIN {X 0,Y 159.168,Z 452.743,A -85,B 0,C 180,E1 -25552.387,E2 -25552.387} C_VEL
LIN {X 0,Y 159.358,Z 452.897,A -85,B 0,C 180,E1 -25558.104,E2 -25558.104} C_VEL
LIN {X 0,Y 160.026,Z 455.669,A -85,B 0,C 180,E1 -25561.887,E2 -25561.887} C_VEL
LIN {X 0,Y 162.158,Z 458.04,A -85,B 0,C 180,E1 -25566.857,E2 -25566.857} C_VEL
LIN {X 0,Y 164.396,Z 461.816,A -85,B 0,C 180,E1 -25570.635,E2 -25570.635} C_VEL
LIN {X 0,Y 165.319,Z 462.965,A -85,B 0,C 180,E1 -25571.883,E2 -25571.883} C_VEL
LIN {X 0,Y 167.842,Z 468.066,A -85,B 0,C 180,E1 -25575.093,E2 -25575.093} C_VEL
LIN {X 0,Y 170.897,Z 474.91,A -85,B 0,C 180,E1 -25578.4,E2 -25578.4} C_VEL
LIN {X 0,Y 174.021,Z 482.239,A -85,B 0,C 180,E1 -25581.313,E2 -25581.313} C_VEL
LIN {X 0,Y 177.769,Z 492.279,A -85,B 0,C 180,E1 -25584.448,E2 -25584.448} C_VEL
LIN {X 0,Y 181.699,Z 504.031,A -85,B 0,C 180,E1 -25587.411,E2 -25587.411} C_VEL
LIN {X 0,Y 182.591,Z 506.978,A -85,B 0,C 180,E1 -25588.053,E2 -25588.053} C_VEL
LIN {X 0,Y 182.904,Z 533.256,A -85,B 0,C 180,E1 -25590.003,E2 -25590.003} C_VEL
LIN {X 0,Y 178.622,Z 582.927,A -85,B 0,C 180,E1 -25591.562,E2 -25591.562} C_VEL
LIN {X 0,Y 176.203,Z 598.152,A -85,B 0,C 180,E1 -25592.32,E2 -25592.32} C_VEL
LIN {X 0,Y 172.602,Z 613.597,A -85,B 0,C 180,E1 -25593.414,E2 -25593.414} C_VEL
LIN {X 0,Y 168.035,Z 628.397,A -85,B 0,C 180,E1 -25594.835,E2 -25594.835} C_VEL
LIN {X 0,Y 163.637,Z 640.323,A -85,B 0,C 180,E1 -25596.362,E2 -25596.362} C_VEL
LIN {X 0,Y 157.541,Z 654.063,A -85,B 0,C 180,E1 -25598.579,E2 -25598.579} C_VEL
